LIN {X 0,Y 300.797,Z 338.167,A -85,B 0,C 180,E1 -24169.506,E2 -24169.506} C_VEL
LIN {X 0,Y 302.211,Z 343.381,A -85,B 0,C 180,E1 -24171.379,E2 -24171.379} C_VEL
LIN {X 0,Y 304.844,Z 348.124,A -85,B 0,C 180,E1 -24171.993,E2 -24171.993} C_VEL
LIN {X 0,Y 312.69,Z 363.044,A -85,B 0,C 180,E1 -24173.748,E2 -24173.748} C_VEL
LIN {X 0,Y 320.446,Z 379.712,A -85,B 0,C 180,E1 -24175.407,E2 -24175.407} C_VEL
LIN {X 0,Y 322.194,Z 383.758,A -85,B 0,C 180,E1 -24175.772,E2 -24175.772} C_VEL
LIN {X 0,Y 326.071,Z 409.314,A -85,B 0,C 180,E1 -24177.018,E2 -24177.018} C_VEL
LIN {X 0,Y 327.432,Z 420.163,A -85,B 0,C 180,E1 -24177.494,E2 -24177.494} C_VEL
LIN {X 0,Y 324.584,Z 482.925,A -85,B 0,C 180,E1 -24178.857,E2 -24178.857} C_VEL
LIN {X 0,Y 323.216,Z 497.454,A -85,B 0,C 180,E1 -24179.389,E2 -24179.389} C_VEL
LIN {X 0,Y 321.164,Z 510.847,A -85,B 0,C 180,E1 -24180.077,E2 -24180.077} C_VEL
LIN {X 0,Y 318.382,Z 524.837,A -85,B 0,C 180,E1 -24181.057,E2 -24181.057} C_VEL
LIN {X 0,Y 315.503,Z 537.338,A -85,B 0,C 180,E1 -24182.215,E2 -24182.215} C_VEL
LIN {X 0,Y 312.38,Z 548.887,A -85,B 0,C 180,E1 -24183.557,E2 -24183.557} C_VEL
LIN {X 0,Y 308.98,Z 560.643,A -85,B 0,C 180,E1 -24185.278,E2 -24185.278} C_VEL
LIN {X 0,Y 305.615,Z 570.588,A -85,B 0,C 180,E1 -24187.073,E2 -24187.073} C_VEL
LIN {X 0,Y 302.649,Z 579.143,A -85,B 0,C 180,E1 -24188.982,E2 -24188.982} C_VEL
LIN {X 0,Y 299.681,Z 587.381,A -85,B 0,C 180,E1 -24191.257,E2 -24191.257} C_VEL
LIN {X 0,Y 297.335,Z 594.052,A -85,B 0,C 180,E1 -24193.583,E2 -24193.583} C_VEL
LIN {X 0,Y 295.224,Z 600.025,A -85,B 0,C 180,E1 -24196.279,E2 -24196.279} C_VEL
LIN {X 0,Y 293.79,Z 604.467,A -85,B 0,C 180,E1 -24199.008,E2 -24199.008} C_VEL
LIN {X 0,Y 292.938,Z 607.496,A -85,B 0,C 180,E1 -24201.755,E2 -24201.755} C_VEL
LIN {X 0,Y 292.769,Z 609.197,A -85,B 0,C 180,E1 -24204.512,E2 -24204.512} C_VEL
LIN {X 0,Y 293.043,Z 609.861,A -85,B 0,C 180,E1 -24206.749,E2 -24206.749} C_VEL
LIN {X 0,Y 292.991,Z 613.677,A -85,B 0,C 180,E1 -24208.633,E2 -24208.633} C_VEL
LIN {X 0,Y 292.914,Z 615.958,A -85,B 0,C 180,E1 -24210.003,E2 -24210.003} C_VEL
LIN {X 0,Y 292.856,Z 617.841,A -85,B 0,C 180,E1 -24211.374,E2 -24211.374} C_VEL
LIN {X 0,Y 292.699,Z 620.456,A -85,B 0,C 180,E1 -24214.12,E2 -24214.12} C_VEL
LIN {X 0,Y 292.878,Z 621.675,A -85,B 0,C 180,E1 -24216.871,E2 -24216.871} C_VEL
LIN {X 0,Y 293.696,Z 621.539,A -85,B 0,C 180,E1 -24219.613,E2 -24219.613} C_VEL
LIN {X 0,Y 295.23,Z 620.064,A -85,B 0,C 180,E1 -24222.332,E2 -24222.332} C_VEL
LIN {X 0,Y 297.448,Z 617.232,A -85,B 0,C 180,E1 -24225.016,E2 -24225.016} C_VEL
LIN {X 0,Y 300.32,Z 613.003,A -85,B 0,C 180,E1 -24227.653,E2 -24227.653} C_VEL
LIN {X 0,Y 304.069,Z 607.239,A -85,B 0,C 180,E1 -24230.218,E2 -24230.218} C_VEL
LIN {X 0,Y 308.257,Z 599.867,A -85,B 0,C 180,E1 -24232.727,E2 -24232.727} C_VEL
LIN {X 0,Y 312.605,Z 591.846,A -85,B 0,C 180,E1 -24234.846,E2 -24234.846} C_VEL
LIN {X 0,Y 317.576,Z 581.993,A -85,B 0,C 180,E1 -24236.885,E2 -24236.885} C_VEL
LIN {X 0,Y 322.111,Z 571.917,A -85,B 0,C 180,E1 -24238.584,E2 -24238.584} C_VEL
LIN {X 0,Y 327.168,Z 559.76,A -85,B 0,C 180,E1 -24240.209,E2 -24240.209} C_VEL
LIN {X 0,Y 331.642,Z 547.568,A -85,B 0,C 180,E1 -24241.519,E2 -24241.519} C_VEL
LIN {X 0,Y 335.963,Z 534.106,A -85,B 0,C 180,E1 -24242.65,E2 -24242.65} C_VEL
LIN {X 0,Y 339.758,Z 520.179,A -85,B 0,C 180,E1 -24243.56,E2 -24243.56} C_VEL
LIN {X 0,Y 343.221,Z 504.513,A -85,B 0,C 180,E1 -24244.32,E2 -24244.32} C_VEL
LIN {X 0,Y 345.995,Z 486.463,A -85,B 0,C 180,E1 -24244.974,E2 -24244.974} C_VEL
LIN {X 0,Y 354.367,Z 425.402,A -85,B 0,C 180,E1 -24246.987,E2 -24246.987} C_VEL
LIN {X 0,Y 354.895,Z 409.778,A -85,B 0,C 180,E1 -24248.063,E2 -24248.063} C_VEL
LIN {X 0,Y 354.892,Z 404.222,A -85,B 0,C 180,E1 -24248.533,E2 -24248.533} C_VEL
LIN {X 0,Y 351.993,Z 398.922,A -85,B 0,C 180,E1 -24250.137,E2 -24250.137} C_VEL
LIN {X 0,Y 349.155,Z 394.154,A -85,B 0,C 180,E1 -24251.973,E2 -24251.973} C_VEL
LIN {X 0,Y 346.445,Z 389.926,A -85,B 0,C 180,E1 -24254.143,E2 -24254.143} C_VEL
LIN {X 0,Y 344.063,Z 386.653,A -85,B 0,C 180,E1 -24256.83,E2 -24256.83} C_VEL
LIN {X 0,Y 342.971,Z 385.018,A -85,B 0,C 180,E1 -24259.085,E2 -24259.085} C_VEL
LIN {X 0,Y 342.569,Z 384.877,A -85,B 0,C 180,E1 -24260.988,E2 -24260.988} C_VEL
LIN {X 0,Y 342.794,Z 385.856,A -85,B 0,C 180,E1 -24263.24,E2 -24263.24} C_VEL
LIN {X 0,Y 343.914,Z 388.274,A -85,B 0,C 180,E1 -24265.709,E2 -24265.709} C_VEL
LIN {X 0,Y 345.45,Z 391.168,A -85,B 0,C 180,E1 -24267.652,E2 -24267.652} C_VEL
LIN {X 0,Y 347.616,Z 395.463,A -85,B 0,C 180,E1 -24269.669,E2 -24269.669} C_VEL
LIN {X 0,Y 350.041,Z 400.682,A -85,B 0,C 180,E1 -24271.488,E2 -24271.488} C_VEL
LIN {X 0,Y 352.53,Z 406.284,A -85,B 0,C 180,E1 -24273.065,E2 -24273.065} C_VEL
LIN {X 0,Y 355.247,Z 413.527,A -85,B 0,C 180,E1 -24274.647,E2 -24274.647} C_VEL
LIN {X 0,Y 355.798,Z 415.257,A -85,B 0,C 180,E1 -24274.963,E2 -24274.963} C_VEL
LIN {X 0,Y 345.082,Z 491.977,A -85,B 0,C 180,E1 -24277.473,E2 -24277.473} C_VEL
LIN {X 0,Y 342.297,Z 506.53,A -85,B 0,C 180,E1 -24278.15,E2 -24278.15} C_VEL
LIN {X 0,Y 339.262,Z 519.363,A -85,B 0,C 180,E1 -24278.939,E2 -24278.939} C_VEL
LIN {X 0,Y 335.283,Z 533.245,A -85,B 0,C 180,E1 -24280.025,E2 -24280.025} C_VEL
LIN {X 0,Y 330.843,Z 546.376,A -85,B 0,C 180,E1 -24281.324,E2 -24281.324} C_VEL
LIN {X 0,Y 326.196,Z 558.349,A -85,B 0,C 180,E1 -24282.827,E2 -24282.827} C_VEL
LIN {X 0,Y 321.417,Z 569.249,A -85,B 0,C 180,E1 -24284.517,E2 -24284.517} C_VEL
LIN {X 0,Y 317.149,Z 578.141,A -85,B 0,C 180,E1 -24286.233,E2 -24286.233} C_VEL
LIN {X 0,Y 312.46,Z 587.071,A -85,B 0,C 180,E1 -24288.36,E2 -24288.36} C_VEL
LIN {X 0,Y 308.831,Z 593.256,A -85,B 0,C 180,E1 -24290.206,E2 -24290.206} C_VEL
LIN {X 0,Y 305.489,Z 598.43,A -85,B 0,C 180,E1 -24292.093,E2 -24292.093} C_VEL
LIN {X 0,Y 301.664,Z 603.858,A -85,B 0,C 180,E1 -24294.671,E2 -24294.671} C_VEL
LIN {X 0,Y 298.589,Z 607.736,A -85,B 0,C 180,E1 -24297.311,E2 -24297.311} C_VEL
LIN {X 0,Y 296.174,Z 610.172,A -85,B 0,C 180,E1 -24300,E2 -24300} C_VEL
LIN {X 0,Y 294.541,Z 611.221,A -85,B 0,C 180,E1 -24302.761,E2 -24302.761} C_VEL
LIN {X 0,Y 293.318,Z 610.914,A -85,B 0,C 180,E1 -24305.481,E2 -24305.481} C_VEL
LIN {X 0,Y 292.619,Z 609.217,A -85,B 0,C 180,E1 -24308.257,E2 -24308.257} C_VEL
LIN {X 0,Y 292.451,Z 606.082,A -85,B 0,C 180,E1 -24311.047,E2 -24311.047} C_VEL
LIN {X 0,Y 292.426,Z 601.359,A -85,B 0,C 180,E1 -24313.859,E2 -24313.859} C_VEL
LIN {X 0,Y 292.682,Z 596.611,A -85,B 0,C 180,E1 -24315.975,E2 -24315.975} C_VEL
LIN {X 0,Y 292.964,Z 589.602,A -85,B 0,C 180,E1 -24318.469,E2 -24318.469} C_VEL
LIN {X 0,Y 293.408,Z 582.124,A -85,B 0,C 180,E1 -24320.617,E2 -24320.617} C_VEL
LIN {X 0,Y 294.017,Z 572.971,A -85,B 0,C 180,E1 -24322.776,E2 -24322.776} C_VEL
LIN {X 0,Y 294.913,Z 561.779,A -85,B 0,C 180,E1 -24324.934,E2 -24324.934} C_VEL
LIN {X 0,Y 295.828,Z 550.441,A -85,B 0,C 180,E1 -24326.735,E2 -24326.735} C_VEL
LIN {X 0,Y 296.868,Z 538.133,A -85,B 0,C 180,E1 -24328.349,E2 -24328.349} C_VEL
LIN {X 0,Y 297.935,Z 524.592,A -85,B 0,C 180,E1 -24329.778,E2 -24329.778} C_VEL
LIN {X 0,Y 298.972,Z 509.581,A -85,B 0,C 180,E1 -24331.026,E2 -24331.026} C_VEL
LIN {X 0,Y 299.875,Z 494.673,A -85,B 0,C 180,E1 -24331.952,E2 -24331.952} C_VEL
LIN {X 0,Y 300.629,Z 479.252,A -85,B 0,C 180,E1 -24332.619,E2 -24332.619} C_VEL
LIN {X 0,Y 304.208,Z 387.346,A -85,B 0,C 180,E1 -24335.809,E2 -24335.809} C_VEL
LIN {X 0,Y 301.045,Z 356.735,A -85,B 0,C 180,E1 -24337.024,E2 -24337.024} C_VEL
LIN {X 0,Y 300.349,Z 346.328,A -85,B 0,C 180,E1 -24337.446,E2 -24337.446} C_VEL
LIN {X 0,Y 300.175,Z 343.352,A -85,B 0,C 180,E1 -24338.04,E2 -24338.04} C_VEL
LIN {X 0,Y 297.01,Z 327.627,A -85,B 0,C 180,E1 -24341.325,E2 -24341.325} C_VEL
LIN {X 0,Y 295.544,Z 320.23,A -85,B 0,C 180,E1 -24342.922,E2 -24342.922} C_VEL
LIN {X 0,Y 295.452,Z 320.238,A -85,B 0,C 180,E1 -24347.302,E2 -24347.302} C_VEL
LIN {X 0,Y 295.445,Z 320.237,A -85,B 0,C 180,E1 -24350.196,E2 -24350.196} C_VEL
LIN {X 0,Y 295.51,Z 320.231,A -85,B 0,C 180,E1 -24353.697,E2 -24353.697} C_VEL
LIN {X 0,Y 295.49,Z 320.226,A -85,B 0,C 180,E1 -24356.958,E2 -24356.958} C_VEL
LIN {X 0,Y 295.495,Z 320.228,A -85,B 0,C 180,E1 -24361.289,E2 -24361.289} C_VEL
LIN {X 0,Y 295.544,Z 320.228,A -85,B 0,C 180,E1 -24364.745,E2 -24364.745} C_VEL
LIN {X 0,Y 295.589,Z 320.223,A -85,B 0,C 180,E1 -24367.716,E2 -24367.716} C_VEL
LIN {X 0,Y 295.64,Z 320.215,A -85,B 0,C 180,E1 -24372.058,E2 -24372.058} C_VEL
LIN {X 0,Y 295.631,Z 320.212,A -85,B 0,C 180,E1 -24372.909,E2 -24372.909} C_VEL
LIN {X 0,Y 296.667,Z 323.105,A -85,B 0,C 180,E1 -24373.079,E2 -24373.079} C_VEL
LIN {X 0,Y 305.844,Z 343.561,A -85,B 0,C 180,E1 -24374.382,E2 -24374.382} C_VEL
LIN {X 0,Y 310.372,Z 356.722,A -85,B 0,C 180,E1 -24375.069,E2 -24375.069} C_VEL
LIN {X 0,Y 307.539,Z 451.607,A -85,B 0,C 180,E1 -24377.25,E2 -24377.25} C_VEL
LIN {X 0,Y 306.788,Z 465.849,A -85,B 0,C 180,E1 -24377.847,E2 -24377.847} C_VEL
LIN {X 0,Y 305.716,Z 479.602,A -85,B 0,C 180,E1 -24378.683,E2 -24378.683} C_VEL
LIN {X 0,Y 304.431,Z 492.441,A -85,B 0,C 180,E1 -24379.725,E2 -24379.725} C_VEL
LIN {X 0,Y 302.99,Z 503.539,A -85,B 0,C 180,E1 -24380.852,E2 -24380.852} C_VEL
LIN {X 0,Y 301.227,Z 515.227,A -85,B 0,C 180,E1 -24382.313,E2 -24382.313} C_VEL
LIN {X 0,Y 299.781,Z 525.862,A -85,B 0,C 180,E1 -24383.961,E2 -24383.961} C_VEL
LIN {X 0,Y 298.014,Z 536.451,A -85,B 0,C 180,E1 -24385.953,E2 -24385.953} C_VEL
LIN {X 0,Y 296.649,Z 545.177,A -85,B 0,C 180,E1 -24387.967,E2 -24387.967} C_VEL
LIN {X 0,Y 295.166,Z 553.586,A -85,B 0,C 180,E1 -24390.337,E2 -24390.337} C_VEL
LIN {X 0,Y 294.481,Z 560.307,A -85,B 0,C 180,E1 -24392.723,E2 -24392.723} C_VEL
LIN {X 0,Y 293.842,Z 564.964,A -85,B 0,C 180,E1 -24394.782,E2 -24394.782} C_VEL
LIN {X 0,Y 293.151,Z 569.825,A -85,B 0,C 180,E1 -24397.548,E2 -24397.548} C_VEL
LIN {X 0,Y 292.981,Z 572.446,A -85,B 0,C 180,E1 -24399.63,E2 -24399.63} C_VEL
LIN {X 0,Y 292.991,Z 574.75,A -85,B 0,C 180,E1 -24402.421,E2 -24402.421} C_VEL
LIN {X 0,Y 293.267,Z 575.703,A -85,B 0,C 180,E1 -24405.228,E2 -24405.228} C_VEL
LIN {X 0,Y 293.998,Z 575.297,A -85,B 0,C 180,E1 -24408.039,E2 -24408.039} C_VEL
LIN {X 0,Y 295.098,Z 573.519,A -85,B 0,C 180,E1 -24410.853,E2 -24410.853} C_VEL
LIN {X 0,Y 296.806,Z 570.267,A -85,B 0,C 180,E1 -24413.649,E2 -24413.649} C_VEL
LIN {X 0,Y 298.986,Z 565.44,A -85,B 0,C 180,E1 -24416.427,E2 -24416.427} C_VEL
LIN {X 0,Y 301.008,Z 560.725,A -85,B 0,C 180,E1 -24418.488,E2 -24418.488} C_VEL
LIN {X 0,Y 303.824,Z 553.8,A -85,B 0,C 180,E1 -24420.857,E2 -24420.857} C_VEL
LIN {X 0,Y 306.53,Z 546.503,A -85,B 0,C 180,E1 -24422.864,E2 -24422.864} C_VEL
LIN {X 0,Y 309.598,Z 537.649,A -85,B 0,C 180,E1 -24424.834,E2 -24424.834} C_VEL
LIN {X 0,Y 312.693,Z 527.837,A -85,B 0,C 180,E1 -24426.608,E2 -24426.608} C_VEL
LIN {X 0,Y 315.695,Z 517.031,A -85,B 0,C 180,E1 -24428.2,E2 -24428.2} C_VEL
LIN {X 0,Y 318.559,Z 505.159,A -85,B 0,C 180,E1 -24429.612,E2 -24429.612} C_VEL
LIN {X 0,Y 321.196,Z 491.982,A -85,B 0,C 180,E1 -24430.856,E2 -24430.856} C_VEL
LIN {X 0,Y 323.29,Z 478.09,A -85,B 0,C 180,E1 -24431.876,E2 -24431.876} C_VEL
LIN {X 0,Y 324.931,Z 464.176,A -85,B 0,C 180,E1 -24432.608,E2 -24432.608} C_VEL
LIN {X 0,Y 325.962,Z 451.27,A -85,B 0,C 180,E1 -24433.075,E2 -24433.075} C_VEL
LIN {X 0,Y 329.077,Z 378.605,A -85,B 0,C 180,E1 -24434.666,E2 -24434.666} C_VEL
LIN {X 0,Y 321.686,Z 362.958,A -85,B 0,C 180,E1 -24436.139,E2 -24436.139} C_VEL
LIN {X 0,Y 315.094,Z 350.798,A -85,B 0,C 180,E1 -24437.49,E2 -24437.49} C_VEL
LIN {X 0,Y 306.413,Z 337.106,A -85,B 0,C 180,E1 -24439.334,E2 -24439.334} C_VEL
LIN {X 0,Y 300.748,Z 328.88,A -85,B 0,C 180,E1 -24440.607,E2 -24440.607} C_VEL
LIN {X 0,Y 298.582,Z 325.449,A -85,B 0,C 180,E1 -24441.125,E2 -24441.125} C_VEL
LIN {X 0,Y 296.267,Z 322.728,A -85,B 0,C 180,E1 -24441.659,E2 -24441.659} C_VEL
LIN {X 0,Y 295.501,Z 320.229,A -85,B 0,C 180,E1 -24441.908,E2 -24441.908} C_VEL
LIN {X 0,Y 295.464,Z 320.215,A -85,B 0,C 180,E1 -24446.064,E2 -24446.064} C_VEL
LIN {X 0,Y 295.486,Z 320.231,A -85,B 0,C 180,E1 -24450.145,E2 -24450.145} C_VEL
LIN {X 0,Y 295.534,Z 320.229,A -85,B 0,C 180,E1 -24454.232,E2 -24454.232} C_VEL
LIN {X 0,Y 295.565,Z 320.215,A -85,B 0,C 180,E1 -24457.717,E2 -24457.717} C_VEL
LIN {X 0,Y 295.598,Z 320.21,A -85,B 0,C 180,E1 -24462.059,E2 -24462.059} C_VEL
LIN {X 0,Y 295.704,Z 320.19,A -85,B 0,C 180,E1 -24466.298,E2 -24466.298} C_VEL
LIN {X 0,Y 295.767,Z 320.183,A -85,B 0,C 180,E1 -24470.458,E2 -24470.458} C_VEL
LIN {X 0,Y 295.98,Z 320.175,A -85,B 0,C 180,E1 -24473.652,E2 -24473.652} C_VEL
LIN {X 0,Y 295.931,Z 320.172,A -85,B 0,C 180,E1 -24474.741,E2 -24474.741} C_VEL
LIN {X 0,Y 295.298,Z 320.24,A -85,B 0,C 180,E1 -24475.878,E2 -24475.878} C_VEL
LIN {X 0,Y 292.497,Z 320.595,A -85,B 0,C 180,E1 -24477.732,E2 -24477.732} C_VEL
LIN {X 0,Y 290.109,Z 320.907,A -85,B 0,C 180,E1 -24479.236,E2 -24479.236} C_VEL
LIN {X 0,Y 289.085,Z 321.022,A -85,B 0,C 180,E1 -24480.401,E2 -24480.401} C_VEL
LIN {X 0,Y 289.003,Z 321.026,A -85,B 0,C 180,E1 -24480.795,E2 -24480.795} C_VEL
LIN {X 0,Y 288.971,Z 321.045,A -85,B 0,C 180,E1 -24484.17,E2 -24484.17} C_VEL
LIN {X 0,Y 288.857,Z 321.038,A -85,B 0,C 180,E1 -24486.964,E2 -24486.964} C_VEL
LIN {X 0,Y 288.675,Z 321.071,A -85,B 0,C 180,E1 -24491.193,E2 -24491.193} C_VEL
LIN {X 0,Y 288.684,Z 321.07,A -85,B 0,C 180,E1 -24494.042,E2 -24494.042} C_VEL
LIN {X 0,Y 288.57,Z 321.083,A -85,B 0,C 180,E1 -24498.814,E2 -24498.814} C_VEL
LIN {X 0,Y 288.493,Z 321.091,A -85,B 0,C 180,E1 -24502.859,E2 -24502.859} C_VEL
LIN {X 0,Y 288.479,Z 321.095,A -85,B 0,C 180,E1 -24506.063,E2 -24506.063} C_VEL
LIN {X 0,Y 288.447,Z 321.1,A -85,B 0,C 180,E1 -24510.661,E2 -24510.661} C_VEL
LIN {X 0,Y 288.455,Z 321.075,A -85,B 0,C 180,E1 -24514.357,E2 -24514.357} C_VEL
LIN {X 0,Y 288.484,Z 321.076,A -85,B 0,C 180,E1 -24517.373,E2 -24517.373} C_VEL
LIN {X 0,Y 288.52,Z 321.266,A -85,B 0,C 180,E1 -24520.841,E2 -24520.841} C_VEL
LIN {X 0,Y 291.2,Z 330.037,A -85,B 0,C 180,E1 -24524.886,E2 -24524.886} C_VEL
LIN {X 0,Y 293.848,Z 339.179,A -85,B 0,C 180,E1 -24528.664,E2 -24528.664} C_VEL
LIN {X 0,Y 294.769,Z 342.618,A -85,B 0,C 180,E1 -24529.975,E2 -24529.975} C_VEL
LIN {X 0,Y 297.416,Z 347.373,A -85,B 0,C 180,E1 -24530.635,E2 -24530.635} C_VEL
LIN {X 0,Y 302.135,Z 355.948,A -85,B 0,C 180,E1 -24531.77,E2 -24531.77} C_VEL
LIN {X 0,Y 307.935,Z 366.963,A -85,B 0,C 180,E1 -24533.1,E2 -24533.1} C_VEL
LIN {X 0,Y 316.042,Z 384.747,A -85,B 0,C 180,E1 -24534.904,E2 -24534.904} C_VEL
LIN {X 0,Y 316.961,Z 387.009,A -85,B 0,C 180,E1 -24535.106,E2 -24535.106} C_VEL
LIN {X 0,Y 320.494,Z 411.032,A -85,B 0,C 180,E1 -24536.3,E2 -24536.3} C_VEL
LIN {X 0,Y 321.741,Z 421.145,A -85,B 0,C 180,E1 -24536.757,E2 -24536.757} C_VEL
LIN {X 0,Y 318.823,Z 482.959,A -85,B 0,C 180,E1 -24538.121,E2 -24538.121} C_VEL
LIN {X 0,Y 317.373,Z 497.579,A -85,B 0,C 180,E1 -24538.67,E2 -24538.67} C_VEL
LIN {X 0,Y 315.072,Z 511.951,A -85,B 0,C 180,E1 -24539.438,E2 -24539.438} C_VEL
LIN {X 0,Y 312.597,Z 523.859,A -85,B 0,C 180,E1 -24540.284,E2 -24540.284} C_VEL
LIN {X 0,Y 309.625,Z 536.466,A -85,B 0,C 180,E1 -24541.456,E2 -24541.456} C_VEL
LIN {X 0,Y 306.392,Z 547.981,A -85,B 0,C 180,E1 -24542.796,E2 -24542.796} C_VEL
LIN {X 0,Y 303.086,Z 559.192,A -85,B 0,C 180,E1 -24544.445,E2 -24544.445} C_VEL
LIN {X 0,Y 299.679,Z 569.096,A -85,B 0,C 180,E1 -24546.226,E2 -24546.226} C_VEL
LIN {X 0,Y 296.488,Z 577.824,A -85,B 0,C 180,E1 -24548.159,E2 -24548.159} C_VEL
LIN {X 0,Y 293.313,Z 586.236,A -85,B 0,C 180,E1 -24550.472,E2 -24550.472} C_VEL
LIN {X 0,Y 291.123,Z 592.138,A -85,B 0,C 180,E1 -24552.501,E2 -24552.501} C_VEL
LIN {X 0,Y 288.819,Z 598.498,A -85,B 0,C 180,E1 -24555.251,E2 -24555.251} C_VEL
LIN {X 0,Y 287.133,Z 603.27,A -85,B 0,C 180,E1 -24558.036,E2 -24558.036} C_VEL
LIN {X 0,Y 286.251,Z 605.853,A -85,B 0,C 180,E1 -24560.141,E2 -24560.141} C_VEL
LIN {X 0,Y 285.656,Z 608.156,A -85,B 0,C 180,E1 -24562.961,E2 -24562.961} C_VEL
LIN {X 0,Y 285.814,Z 609.158,A -85,B 0,C 180,E1 -24565.787,E2 -24565.787} C_VEL
LIN {X 0,Y 285.986,Z 609.357,A -85,B 0,C 180,E1 -24566.932,E2 -24566.932} C_VEL
LIN {X 0,Y 285.926,Z 614.016,A -85,B 0,C 180,E1 -24569.302,E2 -24569.302} C_VEL
LIN {X 0,Y 285.81,Z 617.126,A -85,B 0,C 180,E1 -24571.408,E2 -24571.408} C_VEL
LIN {X 0,Y 285.62,Z 619.941,A -85,B 0,C 180,E1 -24574.222,E2 -24574.222} C_VEL
LIN {X 0,Y 285.81,Z 621.356,A -85,B 0,C 180,E1 -24577.042,E2 -24577.042} C_VEL
LIN {X 0,Y 286.694,Z 621.438,A -85,B 0,C 180,E1 -24579.851,E2 -24579.851} C_VEL
LIN {X 0,Y 288.302,Z 620.193,A -85,B 0,C 180,E1 -24582.634,E2 -24582.634} C_VEL
LIN {X 0,Y 290.678,Z 617.546,A -85,B 0,C 180,E1 -24585.446,E2 -24585.446} C_VEL
LIN {X 0,Y 293.616,Z 613.677,A -85,B 0,C 180,E1 -24588.07,E2 -24588.07} C_VEL
LIN {X 0,Y 296.423,Z 609.715,A -85,B 0,C 180,E1 -24590.041,E2 -24590.041} C_VEL
LIN {X 0,Y 300.744,Z 603.088,A -85,B 0,C 180,E1 -24592.603,E2 -24592.603} C_VEL
LIN {X 0,Y 305.017,Z 595.837,A -85,B 0,C 180,E1 -24594.781,E2 -24594.781} C_VEL
LIN {X 0,Y 309.944,Z 587,A -85,B 0,C 180,E1 -24596.874,E2 -24596.874} C_VEL
LIN {X 0,Y 315.313,Z 576.224,A -85,B 0,C 180,E1 -24598.895,E2 -24598.895} C_VEL
LIN {X 0,Y 320.451,Z 565.032,A -85,B 0,C 180,E1 -24600.547,E2 -24600.547} C_VEL
LIN {X 0,Y 325.459,Z 552.766,A -85,B 0,C 180,E1 -24602.007,E2 -24602.007} C_VEL
LIN {X 0,Y 329.801,Z 540.581,A -85,B 0,C 180,E1 -24603.157,E2 -24603.157} C_VEL
LIN {X 0,Y 334.437,Z 525.531,A -85,B 0,C 180,E1 -24604.257,E2 -24604.257} C_VEL
LIN {X 0,Y 337.971,Z 511.719,A -85,B 0,C 180,E1 -24605.02,E2 -24605.02} C_VEL
LIN {X 0,Y 341.055,Z 495.588,A -85,B 0,C 180,E1 -24605.693,E2 -24605.693} C_VEL
LIN {X 0,Y 350.969,Z 427.139,A -85,B 0,C 180,E1 -24607.962,E2 -24607.962} C_VEL
LIN {X 0,Y 351.68,Z 411.85,A -85,B 0,C 180,E1 -24609.034,E2 -24609.034} C_VEL
LIN {X 0,Y 351.667,Z 409.048,A -85,B 0,C 180,E1 -24609.298,E2 -24609.298} C_VEL
LIN {X 0,Y 348.159,Z 402.533,A -85,B 0,C 180,E1 -24611.481,E2 -24611.481} C_VEL
LIN {X 0,Y 345.228,Z 397.709,A -85,B 0,C 180,E1 -24613.748,E2 -24613.748} C_VEL
LIN {X 0,Y 343.498,Z 395.172,A -85,B 0,C 180,E1 -24615.483,E2 -24615.483} C_VEL
LIN {X 0,Y 341.777,Z 392.491,A -85,B 0,C 180,E1 -24618.134,E2 -24618.134} C_VEL
LIN {X 0,Y 341.305,Z 391.878,A -85,B 0,C 180,E1 -24619.409,E2 -24619.409} C_VEL
LIN {X 0,Y 340.993,Z 391.879,A -85,B 0,C 180,E1 -24621.316,E2 -24621.316} C_VEL
LIN {X 0,Y 341.332,Z 393.124,A -85,B 0,C 180,E1 -24623.65,E2 -24623.65} C_VEL
LIN {X 0,Y 342.426,Z 395.587,A -85,B 0,C 180,E1 -24625.902,E2 -24625.902} C_VEL
LIN {X 0,Y 343.605,Z 397.91,A -85,B 0,C 180,E1 -24627.436,E2 -24627.436} C_VEL
LIN {X 0,Y 345.579,Z 402.063,A -85,B 0,C 180,E1 -24629.381,E2 -24629.381} C_VEL
LIN {X 0,Y 347.724,Z 407.035,A -85,B 0,C 180,E1 -24631.117,E2 -24631.117} C_VEL
LIN {X 0,Y 349.782,Z 411.933,A -85,B 0,C 180,E1 -24632.523,E2 -24632.523} C_VEL
LIN {X 0,Y 352.218,Z 418.848,A -85,B 0,C 180,E1 -24634.055,E2 -24634.055} C_VEL
LIN {X 0,Y 341.436,Z 492.23,A -85,B 0,C 180,E1 -24636.46,E2 -24636.46} C_VEL
LIN {X 0,Y 338.396,Z 507.306,A -85,B 0,C 180,E1 -24637.163,E2 -24637.163} C_VEL
LIN {X 0,Y 335.364,Z 519.52,A -85,B 0,C 180,E1 -24637.917,E2 -24637.917} C_VEL
LIN {X 0,Y 331.412,Z 532.712,A -85,B 0,C 180,E1 -24638.943,E2 -24638.943} C_VEL
LIN {X 0,Y 326.679,Z 546.19,A -85,B 0,C 180,E1 -24640.263,E2 -24640.263} C_VEL
LIN {X 0,Y 322.237,Z 557.207,A -85,B 0,C 180,E1 -24641.628,E2 -24641.628} C_VEL
LIN {X 0,Y 317.17,Z 568.297,A -85,B 0,C 180,E1 -24643.316,E2 -24643.316} C_VEL
LIN {X 0,Y 311.931,Z 578.669,A -85,B 0,C 180,E1 -24645.313,E2 -24645.313} C_VEL
LIN {X 0,Y 306.938,Z 587.578,A -85,B 0,C 180,E1 -24647.479,E2 -24647.479} C_VEL
LIN {X 0,Y 303.122,Z 593.711,A -85,B 0,C 180,E1 -24649.347,E2 -24649.347} C_VEL
LIN {X 0,Y 299.597,Z 598.81,A -85,B 0,C 180,E1 -24651.259,E2 -24651.259} C_VEL
LIN {X 0,Y 296.157,Z 603.344,A -85,B 0,C 180,E1 -24653.408,E2 -24653.408} C_VEL
LIN {X 0,Y 292.946,Z 607.163,A -85,B 0,C 180,E1 -24655.887,E2 -24655.887} C_VEL
LIN {X 0,Y 290.12,Z 609.911,A -85,B 0,C 180,E1 -24658.617,E2 -24658.617} C_VEL
LIN {X 0,Y 288.146,Z 611.271,A -85,B 0,C 180,E1 -24661.393,E2 -24661.393} C_VEL
LIN {X 0,Y 286.718,Z 611.295,A -85,B 0,C 180,E1 -24664.203,E2 -24664.203} C_VEL
LIN {X 0,Y 285.743,Z 609.949,A -85,B 0,C 180,E1 -24667.04,E2 -24667.04} C_VEL
LIN {X 0,Y 285.4,Z 607.188,A -85,B 0,C 180,E1 -24669.892,E2 -24669.892} C_VEL
LIN {X 0,Y 285.3,Z 604.08,A -85,B 0,C 180,E1 -24672.045,E2 -24672.045} C_VEL
LIN {X 0,Y 285.384,Z 600.038,A -85,B 0,C 180,E1 -24674.208,E2 -24674.208} C_VEL
LIN {X 0,Y 285.636,Z 595.097,A -85,B 0,C 180,E1 -24676.332,E2 -24676.332} C_VEL
LIN {X 0,Y 285.991,Z 587.465,A -85,B 0,C 180,E1 -24678.936,E2 -24678.936} C_VEL
LIN {X 0,Y 286.496,Z 579.493,A -85,B 0,C 180,E1 -24681.138,E2 -24681.138} C_VEL
LIN {X 0,Y 287.123,Z 569.762,A -85,B 0,C 180,E1 -24683.355,E2 -24683.355} C_VEL
LIN {X 0,Y 288.023,Z 558.97,A -85,B 0,C 180,E1 -24685.38,E2 -24685.38} C_VEL
LIN {X 0,Y 289.01,Z 547.131,A -85,B 0,C 180,E1 -24687.203,E2 -24687.203} C_VEL
LIN {X 0,Y 290.123,Z 533.856,A -85,B 0,C 180,E1 -24688.872,E2 -24688.872} C_VEL
LIN {X 0,Y 291.149,Z 520.473,A -85,B 0,C 180,E1 -24690.227,E2 -24690.227} C_VEL
LIN {X 0,Y 292.111,Z 506.469,A -85,B 0,C 180,E1 -24691.335,E2 -24691.335} C_VEL
LIN {X 0,Y 293.096,Z 490.523,A -85,B 0,C 180,E1 -24692.274,E2 -24692.274} C_VEL
LIN {X 0,Y 293.959,Z 468.714,A -85,B 0,C 180,E1 -24693.131,E2 -24693.131} C_VEL
LIN {X 0,Y 297.198,Z 387.774,A -85,B 0,C 180,E1 -24696.028,E2 -24696.028} C_VEL
LIN {X 0,Y 293.975,Z 356.014,A -85,B 0,C 180,E1 -24697.32,E2 -24697.32} C_VEL
LIN {X 0,Y 293.437,Z 346.313,A -85,B 0,C 180,E1 -24697.744,E2 -24697.744} C_VEL
LIN {X 0,Y 290.656,Z 331.948,A -85,B 0,C 180,E1 -24700.779,E2 -24700.779} C_VEL
LIN {X 0,Y 288.517,Z 321.104,A -85,B 0,C 180,E1 -24703.135,E2 -24703.135} C_VEL
LIN {X 0,Y 288.403,Z 321.116,A -85,B 0,C 180,E1 -24707.15,E2 -24707.15} C_VEL
LIN {X 0,Y 288.4,Z 321.116,A -85,B 0,C 180,E1 -24711.004,E2 -24711.004} C_VEL
LIN {X 0,Y 288.422,Z 321.107,A -85,B 0,C 180,E1 -24714.345,E2 -24714.345} C_VEL
LIN {X 0,Y 288.433,Z 321.112,A -85,B 0,C 180,E1 -24718.207,E2 -24718.207} C_VEL
LIN {X 0,Y 288.476,Z 321.099,A -85,B 0,C 180,E1 -24722.523,E2 -24722.523} C_VEL
LIN {X 0,Y 288.466,Z 321.11,A -85,B 0,C 180,E1 -24725.617,E2 -24725.617} C_VEL
LIN {X 0,Y 288.514,Z 321.104,A -85,B 0,C 180,E1 -24728.641,E2 -24728.641} C_VEL
LIN {X 0,Y 288.598,Z 321.09,A -85,B 0,C 180,E1 -24732.28,E2 -24732.28} C_VEL
LIN {X 0,Y 289.663,Z 324.032,A -85,B 0,C 180,E1 -24732.467,E2 -24732.467} C_VEL
LIN {X 0,Y 299.147,Z 344.931,A -85,B 0,C 180,E1 -24733.863,E2 -24733.863} C_VEL
LIN {X 0,Y 303.714,Z 357.761,A -85,B 0,C 180,E1 -24734.569,E2 -24734.569} C_VEL
LIN {X 0,Y 300.953,Z 451.074,A -85,B 0,C 180,E1 -24736.752,E2 -24736.752} C_VEL
LIN {X 0,Y 300.112,Z 465.674,A -85,B 0,C 180,E1 -24737.358,E2 -24737.358} C_VEL
LIN {X 0,Y 299.123,Z 478.993,A -85,B 0,C 180,E1 -24738.174,E2 -24738.174} C_VEL
LIN {X 0,Y 297.88,Z 491.182,A -85,B 0,C 180,E1 -24739.154,E2 -24739.154} C_VEL
LIN {X 0,Y 296.416,Z 502.592,A -85,B 0,C 180,E1 -24740.304,E2 -24740.304} C_VEL
LIN {X 0,Y 294.57,Z 514.523,A -85,B 0,C 180,E1 -24741.794,E2 -24741.794} C_VEL
LIN {X 0,Y 293.043,Z 525.348,A -85,B 0,C 180,E1 -24743.478,E2 -24743.478} C_VEL
LIN {X 0,Y 291.527,Z 534.46,A -85,B 0,C 180,E1 -24745.173,E2 -24745.173} C_VEL
LIN {X 0,Y 289.955,Z 543.602,A -85,B 0,C 180,E1 -24747.227,E2 -24747.227} C_VEL
LIN {X 0,Y 288.583,Z 551.237,A -85,B 0,C 180,E1 -24749.301,E2 -24749.301} C_VEL
LIN {X 0,Y 287.813,Z 557.557,A -85,B 0,C 180,E1 -24751.391,E2 -24751.391} C_VEL
LIN {X 0,Y 287.156,Z 562.775,A -85,B 0,C 180,E1 -24753.493,E2 -24753.493} C_VEL
LIN {X 0,Y 286.337,Z 568.329,A -85,B 0,C 180,E1 -24756.316,E2 -24756.316} C_VEL
LIN {X 0,Y 285.958,Z 571.43,A -85,B 0,C 180,E1 -24758.448,E2 -24758.448} C_VEL
LIN {X 0,Y 285.914,Z 574.494,A -85,B 0,C 180,E1 -24761.496,E2 -24761.496} C_VEL
LIN {X 0,Y 286.026,Z 575.882,A -85,B 0,C 180,E1 -24764.171,E2 -24764.171} C_VEL
LIN {X 0,Y 286.62,Z 576.071,A -85,B 0,C 180,E1 -24767.049,E2 -24767.049} C_VEL
LIN {X 0,Y 287.576,Z 574.891,A -85,B 0,C 180,E1 -24769.934,E2 -24769.934} C_VEL
LIN {X 0,Y 289.128,Z 572.273,A -85,B 0,C 180,E1 -24772.802,E2 -24772.802} C_VEL
LIN {X 0,Y 291.197,Z 568.15,A -85,B 0,C 180,E1 -24775.652,E2 -24775.652} C_VEL
LIN {X 0,Y 293.811,Z 562.39,A -85,B 0,C 180,E1 -24778.472,E2 -24778.472} C_VEL
LIN {X 0,Y 296.64,Z 555.823,A -85,B 0,C 180,E1 -24780.898,E2 -24780.898} C_VEL
LIN {X 0,Y 299.885,Z 547.587,A -85,B 0,C 180,E1 -24783.286,E2 -24783.286} C_VEL
LIN {X 0,Y 303.037,Z 538.876,A -85,B 0,C 180,E1 -24785.295,E2 -24785.295} C_VEL
LIN {X 0,Y 305.936,Z 530.186,A -85,B 0,C 180,E1 -24786.937,E2 -24786.937} C_VEL
LIN {X 0,Y 309.307,Z 518.619,A -85,B 0,C 180,E1 -24788.72,E2 -24788.72} C_VEL
LIN {X 0,Y 312.387,Z 506.521,A -85,B 0,C 180,E1 -24790.204,E2 -24790.204} C_VEL
LIN {X 0,Y 314.997,Z 494.177,A -85,B 0,C 180,E1 -24791.412,E2 -24791.412} C_VEL
LIN {X 0,Y 317.142,Z 480.787,A -85,B 0,C 180,E1 -24792.45,E2 -24792.45} C_VEL
LIN {X 0,Y 318.992,Z 466.368,A -85,B 0,C 180,E1 -24793.262,E2 -24793.262} C_VEL
LIN {X 0,Y 320.198,Z 452.251,A -85,B 0,C 180,E1 -24793.802,E2 -24793.802} C_VEL
LIN {X 0,Y 323.423,Z 380.829,A -85,B 0,C 180,E1 -24795.384,E2 -24795.384} C_VEL
LIN {X 0,Y 316.028,Z 365.317,A -85,B 0,C 180,E1 -24796.915,E2 -24796.915} C_VEL
LIN {X 0,Y 310.501,Z 355.137,A -85,B 0,C 180,E1 -24798.093,E2 -24798.093} C_VEL
LIN {X 0,Y 302.397,Z 342.254,A -85,B 0,C 180,E1 -24799.873,E2 -24799.873} C_VEL
LIN {X 0,Y 296.243,Z 333.323,A -85,B 0,C 180,E1 -24801.305,E2 -24801.305} C_VEL
LIN {X 0,Y 294.19,Z 330.234,A -85,B 0,C 180,E1 -24801.808,E2 -24801.808} C_VEL
LIN {X 0,Y 292.018,Z 327.194,A -85,B 0,C 180,E1 -24802.345,E2 -24802.345} C_VEL
LIN {X 0,Y 291.225,Z 325.908,A -85,B 0,C 180,E1 -24802.551,E2 -24802.551} C_VEL
LIN {X 0,Y 289.971,Z 324.694,A -85,B 0,C 180,E1 -24802.851,E2 -24802.851} C_VEL
LIN {X 0,Y 288.642,Z 322.163,A -85,B 0,C 180,E1 -24803.218,E2 -24803.218} C_VEL
LIN {X 0,Y 288.433,Z 321.081,A -85,B 0,C 180,E1 -24803.328,E2 -24803.328} C_VEL
LIN {X 0,Y 288.427,Z 321.091,A -85,B 0,C 180,E1 -24806.044,E2 -24806.044} C_VEL
LIN {X 0,Y 288.437,Z 321.103,A -85,B 0,C 180,E1 -24809.338,E2 -24809.338} C_VEL
LIN {X 0,Y 288.463,Z 321.097,A -85,B 0,C 180,E1 -24812.525,E2 -24812.525} C_VEL
LIN {X 0,Y 288.464,Z 321.102,A -85,B 0,C 180,E1 -24815.62,E2 -24815.62} C_VEL
LIN {X 0,Y 288.488,Z 321.108,A -85,B 0,C 180,E1 -24818.642,E2 -24818.642} C_VEL
LIN {X 0,Y 288.551,Z 321.084,A -85,B 0,C 180,E1 -24821.605,E2 -24821.605} C_VEL
LIN {X 0,Y 288.641,Z 321.069,A -85,B 0,C 180,E1 -24826.073,E2 -24826.073} C_VEL
LIN {X 0,Y 288.718,Z 321.062,A -85,B 0,C 180,E1 -24830.222,E2 -24830.222} C_VEL
LIN {X 0,Y 288.887,Z 321.055,A -85,B 0,C 180,E1 -24834.434,E2 -24834.434} C_VEL
LIN {X 0,Y 288.934,Z 321.033,A -85,B 0,C 180,E1 -24837.221,E2 -24837.221} C_VEL
LIN {X 0,Y 289.003,Z 321.026,A -85,B 0,C 180,E1 -24840.795,E2 -24840.795} C_VEL
LIN {X 0,Y 288.342,Z 321.106,A -85,B 0,C 180,E1 -24841.958,E2 -24841.958} C_VEL
LIN {X 0,Y 285.487,Z 321.476,A -85,B 0,C 180,E1 -24843.85,E2 -24843.85} C_VEL
LIN {X 0,Y 283.028,Z 321.782,A -85,B 0,C 180,E1 -24845.386,E2 -24845.386} C_VEL
LIN {X 0,Y 281.925,Z 321.905,A -85,B 0,C 180,E1 -24846.577,E2 -24846.577} C_VEL
LIN {X 0,Y 281.809,Z 321.916,A -85,B 0,C 180,E1 -24846.981,E2 -24846.981} C_VEL
LIN {X 0,Y 281.618,Z 321.945,A -85,B 0,C 180,E1 -24851.477,E2 -24851.477} C_VEL
LIN {X 0,Y 281.604,Z 321.957,A -85,B 0,C 180,E1 -24854.403,E2 -24854.403} C_VEL
LIN {X 0,Y 281.517,Z 321.964,A -85,B 0,C 180,E1 -24859.02,E2 -24859.02} C_VEL
LIN {X 0,Y 281.432,Z 321.976,A -85,B 0,C 180,E1 -24863.467,E2 -24863.467} C_VEL
LIN {X 0,Y 281.408,Z 321.975,A -85,B 0,C 180,E1 -24866.618,E2 -24866.618} C_VEL
LIN {X 0,Y 281.384,Z 321.982,A -85,B 0,C 180,E1 -24869.858,E2 -24869.858} C_VEL
LIN {X 0,Y 281.381,Z 321.979,A -85,B 0,C 180,E1 -24873.206,E2 -24873.206} C_VEL
LIN {X 0,Y 281.447,Z 321.949,A -85,B 0,C 180,E1 -24877.22,E2 -24877.22} C_VEL
LIN {X 0,Y 281.468,Z 322.099,A -85,B 0,C 180,E1 -24879.46,E2 -24879.46} C_VEL
LIN {X 0,Y 284.15,Z 330.711,A -85,B 0,C 180,E1 -24883.647,E2 -24883.647} C_VEL
LIN {X 0,Y 286.486,Z 338.767,A -85,B 0,C 180,E1 -24887.179,E2 -24887.179} C_VEL
LIN {X 0,Y 287.478,Z 342.144,A -85,B 0,C 180,E1 -24888.501,E2 -24888.501} C_VEL
LIN {X 0,Y 289.985,Z 346.644,A -85,B 0,C 180,E1 -24889.172,E2 -24889.172} C_VEL
LIN {X 0,Y 294.715,Z 354.806,A -85,B 0,C 180,E1 -24890.377,E2 -24890.377} C_VEL
LIN {X 0,Y 301.598,Z 367.687,A -85,B 0,C 180,E1 -24892.05,E2 -24892.05} C_VEL
LIN {X 0,Y 308.041,Z 381.411,A -85,B 0,C 180,E1 -24893.559,E2 -24893.559} C_VEL
LIN {X 0,Y 311.778,Z 390.361,A -85,B 0,C 180,E1 -24894.42,E2 -24894.42} C_VEL
LIN {X 0,Y 315.111,Z 413.914,A -85,B 0,C 180,E1 -24895.612,E2 -24895.612} C_VEL
LIN {X 0,Y 316.106,Z 422.6,A -85,B 0,C 180,E1 -24896.006,E2 -24896.006} C_VEL
LIN {X 0,Y 313.195,Z 482.218,A -85,B 0,C 180,E1 -24897.336,E2 -24897.336} C_VEL
LIN {X 0,Y 311.784,Z 496.199,A -85,B 0,C 180,E1 -24897.853,E2 -24897.853} C_VEL
LIN {X 0,Y 309.625,Z 509.697,A -85,B 0,C 180,E1 -24898.556,E2 -24898.556} C_VEL
LIN {X 0,Y 306.893,Z 522.877,A -85,B 0,C 180,E1 -24899.485,E2 -24899.485} C_VEL
LIN {X 0,Y 303.808,Z 535.594,A -85,B 0,C 180,E1 -24900.668,E2 -24900.668} C_VEL
LIN {X 0,Y 300.126,Z 548.355,A -85,B 0,C 180,E1 -24902.18,E2 -24902.18} C_VEL
LIN {X 0,Y 297.008,Z 558.497,A -85,B 0,C 180,E1 -24903.701,E2 -24903.701} C_VEL
LIN {X 0,Y 293.198,Z 569.229,A -85,B 0,C 180,E1 -24905.667,E2 -24905.667} C_VEL
LIN {X 0,Y 289.406,Z 579.166,A -85,B 0,C 180,E1 -24907.971,E2 -24907.971} C_VEL
LIN {X 0,Y 286.208,Z 587.22,A -85,B 0,C 180,E1 -24910.34,E2 -24910.34} C_VEL
LIN {X 0,Y 283.676,Z 593.753,A -85,B 0,C 180,E1 -24912.768,E2 -24912.768} C_VEL
LIN {X 0,Y 281.394,Z 599.601,A -85,B 0,C 180,E1 -24915.59,E2 -24915.59} C_VEL
LIN {X 0,Y 279.834,Z 603.927,A -85,B 0,C 180,E1 -24918.452,E2 -24918.452} C_VEL
LIN {X 0,Y 278.828,Z 606.846,A -85,B 0,C 180,E1 -24921.335,E2 -24921.335} C_VEL
LIN {X 0,Y 278.589,Z 608.442,A -85,B 0,C 180,E1 -24924.232,E2 -24924.232} C_VEL
LIN {X 0,Y 278.95,Z 608.814,A -85,B 0,C 180,E1 -24927.125,E2 -24927.125} C_VEL
LIN {X 0,Y 278.901,Z 613.084,A -85,B 0,C 180,E1 -24929.284,E2 -24929.284} C_VEL
LIN {X 0,Y 278.748,Z 616.401,A -85,B 0,C 180,E1 -24931.443,E2 -24931.443} C_VEL
LIN {X 0,Y 278.552,Z 619.411,A -85,B 0,C 180,E1 -24934.33,E2 -24934.33} C_VEL
LIN {X 0,Y 278.746,Z 621.033,A -85,B 0,C 180,E1 -24937.221,E2 -24937.221} C_VEL
LIN {X 0,Y 279.7,Z 621.333,A -85,B 0,C 180,E1 -24940.099,E2 -24940.099} C_VEL
LIN {X 0,Y 281.385,Z 620.316,A -85,B 0,C 180,E1 -24942.949,E2 -24942.949} C_VEL
LIN {X 0,Y 283.777,Z 617.981,A -85,B 0,C 180,E1 -24945.758,E2 -24945.758} C_VEL
LIN {X 0,Y 286.897,Z 614.293,A -85,B 0,C 180,E1 -24948.508,E2 -24948.508} C_VEL
LIN {X 0,Y 290.929,Z 609.151,A -85,B 0,C 180,E1 -24951.174,E2 -24951.174} C_VEL
LIN {X 0,Y 295.45,Z 602.478,A -85,B 0,C 180,E1 -24953.771,E2 -24953.771} C_VEL
LIN {X 0,Y 300.095,Z 595.153,A -85,B 0,C 180,E1 -24955.956,E2 -24955.956} C_VEL
LIN {X 0,Y 305.382,Z 586.197,A -85,B 0,C 180,E1 -24958.051,E2 -24958.051} C_VEL
LIN {X 0,Y 310.187,Z 577.054,A -85,B 0,C 180,E1 -24959.791,E2 -24959.791} C_VEL
LIN {X 0,Y 315.524,Z 566.119,A -85,B 0,C 180,E1 -24961.448,E2 -24961.448} C_VEL
LIN {X 0,Y 320.708,Z 554.133,A -85,B 0,C 180,E1 -24962.91,E2 -24962.91} C_VEL
LIN {X 0,Y 325.204,Z 542.381,A -85,B 0,C 180,E1 -24964.059,E2 -24964.059} C_VEL
LIN {X 0,Y 329.988,Z 527.924,A -85,B 0,C 180,E1 -24965.156,E2 -24965.156} C_VEL
LIN {X 0,Y 333.918,Z 513.682,A -85,B 0,C 180,E1 -24965.972,E2 -24965.972} C_VEL
LIN {X 0,Y 337.119,Z 498.652,A -85,B 0,C 180,E1 -24966.637,E2 -24966.637} C_VEL
LIN {X 0,Y 347.814,Z 428.371,A -85,B 0,C 180,E1 -24968.993,E2 -24968.993} C_VEL
LIN {X 0,Y 348.627,Z 414.553,A -85,B 0,C 180,E1 -24969.984,E2 -24969.984} C_VEL
LIN {X 0,Y 348.39,Z 413.598,A -85,B 0,C 180,E1 -24970.182,E2 -24970.182} C_VEL
LIN {X 0,Y 345.407,Z 407.997,A -85,B 0,C 180,E1 -24972.226,E2 -24972.226} C_VEL
LIN {X 0,Y 342.932,Z 403.75,A -85,B 0,C 180,E1 -24974.366,E2 -24974.366} C_VEL
LIN {X 0,Y 341.197,Z 401.173,A -85,B 0,C 180,E1 -24976.337,E2 -24976.337} C_VEL
LIN {X 0,Y 339.928,Z 399.07,A -85,B 0,C 180,E1 -24978.747,E2 -24978.747} C_VEL
LIN {X 0,Y 339.529,Z 398.691,A -85,B 0,C 180,E1 -24980.243,E2 -24980.243} C_VEL
LIN {X 0,Y 339.492,Z 399.313,A -85,B 0,C 180,E1 -24982.556,E2 -24982.556} C_VEL
LIN {X 0,Y 340.265,Z 401.392,A -85,B 0,C 180,E1 -24984.955,E2 -24984.955} C_VEL
LIN {X 0,Y 341.695,Z 404.431,A -85,B 0,C 180,E1 -24987.099,E2 -24987.099} C_VEL
LIN {X 0,Y 343.49,Z 408.531,A -85,B 0,C 180,E1 -24989.038,E2 -24989.038} C_VEL
LIN {X 0,Y 345.35,Z 413.087,A -85,B 0,C 180,E1 -24990.646,E2 -24990.646} C_VEL
LIN {X 0,Y 347.183,Z 417.736,A -85,B 0,C 180,E1 -24992.004,E2 -24992.004} C_VEL
LIN {X 0,Y 348.748,Z 422.526,A -85,B 0,C 180,E1 -24993.106,E2 -24993.106} C_VEL
LIN {X 0,Y 337.922,Z 492.892,A -85,B 0,C 180,E1 -24995.427,E2 -24995.427} C_VEL
LIN {X 0,Y 334.622,Z 508.364,A -85,B 0,C 180,E1 -24996.155,E2 -24996.155} C_VEL
LIN {X 0,Y 331.219,Z 521.24,A -85,B 0,C 180,E1 -24996.969,E2 -24996.969} C_VEL
LIN {X 0,Y 327.11,Z 534.131,A -85,B 0,C 180,E1 -24997.992,E2 -24997.992} C_VEL
LIN {X 0,Y 322.357,Z 546.934,A -85,B 0,C 180,E1 -24999.27,E2 -24999.27} C_VEL
LIN {X 0,Y 317.562,Z 558.153,A -85,B 0,C 180,E1 -25000.679,E2 -25000.679} C_VEL
LIN {X 0,Y 312.256,Z 569.112,A -85,B 0,C 180,E1 -25002.372,E2 -25002.372} C_VEL
LIN {X 0,Y 307.412,Z 578.201,A -85,B 0,C 180,E1 -25004.132,E2 -25004.132} C_VEL
LIN {X 0,Y 302.232,Z 587.003,A -85,B 0,C 180,E1 -25006.258,E2 -25006.258} C_VEL
LIN {X 0,Y 297.494,Z 594.217,A -85,B 0,C 180,E1 -25008.455,E2 -25008.455} C_VEL
LIN {X 0,Y 292.61,Z 600.721,A -85,B 0,C 180,E1 -25011.049,E2 -25011.049} C_VEL
LIN {X 0,Y 289.249,Z 604.751,A -85,B 0,C 180,E1 -25013.167,E2 -25013.167} C_VEL
LIN {X 0,Y 285.855,Z 608.307,A -85,B 0,C 180,E1 -25015.784,E2 -25015.784} C_VEL
LIN {X 0,Y 282.98,Z 610.633,A -85,B 0,C 180,E1 -25018.582,E2 -25018.582} C_VEL
LIN {X 0,Y 280.992,Z 611.605,A -85,B 0,C 180,E1 -25021.428,E2 -25021.428} C_VEL
LIN {X 0,Y 279.57,Z 611.242,A -85,B 0,C 180,E1 -25024.311,E2 -25024.311} C_VEL
LIN {X 0,Y 278.602,Z 609.508,A -85,B 0,C 180,E1 -25027.222,E2 -25027.222} C_VEL
LIN {X 0,Y 278.324,Z 606.364,A -85,B 0,C 180,E1 -25030.146,E2 -25030.146} C_VEL
LIN {X 0,Y 278.216,Z 602.974,A -85,B 0,C 180,E1 -25032.357,E2 -25032.357} C_VEL
LIN {X 0,Y 278.346,Z 598.644,A -85,B 0,C 180,E1 -25034.575,E2 -25034.575} C_VEL
LIN {X 0,Y 278.67,Z 592.02,A -85,B 0,C 180,E1 -25037.218,E2 -25037.218} C_VEL
LIN {X 0,Y 279.102,Z 583.858,A -85,B 0,C 180,E1 -25039.804,E2 -25039.804} C_VEL
LIN {X 0,Y 279.664,Z 575.096,A -85,B 0,C 180,E1 -25042.067,E2 -25042.067} C_VEL
LIN {X 0,Y 280.461,Z 564.396,A -85,B 0,C 180,E1 -25044.336,E2 -25044.336} C_VEL
LIN {X 0,Y 281.315,Z 553.835,A -85,B 0,C 180,E1 -25046.179,E2 -25046.179} C_VEL
LIN {X 0,Y 282.341,Z 541.795,A -85,B 0,C 180,E1 -25047.921,E2 -25047.921} C_VEL
LIN {X 0,Y 283.349,Z 529.114,A -85,B 0,C 180,E1 -25049.427,E2 -25049.427} C_VEL
LIN {X 0,Y 284.301,Z 516.349,A -85,B 0,C 180,E1 -25050.655,E2 -25050.655} C_VEL
LIN {X 0,Y 285.35,Z 501.786,A -85,B 0,C 180,E1 -25051.751,E2 -25051.751} C_VEL
LIN {X 0,Y 286.24,Z 486.687,A -85,B 0,C 180,E1 -25052.572,E2 -25052.572} C_VEL
LIN {X 0,Y 290.117,Z 387.677,A -85,B 0,C 180,E1 -25056.268,E2 -25056.268} C_VEL
LIN {X 0,Y 287.033,Z 356.83,A -85,B 0,C 180,E1 -25057.56,E2 -25057.56} C_VEL
LIN {X 0,Y 286.359,Z 346.613,A -85,B 0,C 180,E1 -25057.99,E2 -25057.99} C_VEL
LIN {X 0,Y 283.076,Z 330.143,A -85,B 0,C 180,E1 -25061.535,E2 -25061.535} C_VEL
LIN {X 0,Y 281.441,Z 321.986,A -85,B 0,C 180,E1 -25063.345,E2 -25063.345} C_VEL
LIN {X 0,Y 281.351,Z 321.995,A -85,B 0,C 180,E1 -25067.76,E2 -25067.76} C_VEL
LIN {X 0,Y 281.335,Z 321.996,A -85,B 0,C 180,E1 -25071.503,E2 -25071.503} C_VEL
LIN {X 0,Y 281.382,Z 321.979,A -85,B 0,C 180,E1 -25075.232,E2 -25075.232} C_VEL
LIN {X 0,Y 281.381,Z 321.993,A -85,B 0,C 180,E1 -25078.479,E2 -25078.479} C_VEL
LIN {X 0,Y 281.411,Z 321.978,A -85,B 0,C 180,E1 -25081.773,E2 -25081.773} C_VEL
LIN {X 0,Y 281.404,Z 321.989,A -85,B 0,C 180,E1 -25084.963,E2 -25084.963} C_VEL
LIN {X 0,Y 281.455,Z 321.984,A -85,B 0,C 180,E1 -25088.078,E2 -25088.078} C_VEL
LIN {X 0,Y 281.585,Z 322.049,A -85,B 0,C 180,E1 -25091.634,E2 -25091.634} C_VEL
LIN {X 0,Y 282.55,Z 324.754,A -85,B 0,C 180,E1 -25091.806,E2 -25091.806} C_VEL
LIN {X 0,Y 291.745,Z 344.76,A -85,B 0,C 180,E1 -25093.214,E2 -25093.214} C_VEL
LIN {X 0,Y 295.697,Z 354.805,A -85,B 0,C 180,E1 -25093.826,E2 -25093.826} C_VEL
LIN {X 0,Y 297.223,Z 359.957,A -85,B 0,C 180,E1 -25094.091,E2 -25094.091} C_VEL
LIN {X 0,Y 294.332,Z 451.614,A -85,B 0,C 180,E1 -25096.273,E2 -25096.273} C_VEL
LIN {X 0,Y 293.477,Z 466.159,A -85,B 0,C 180,E1 -25096.892,E2 -25096.892} C_VEL
LIN {X 0,Y 292.432,Z 479.469,A -85,B 0,C 180,E1 -25097.723,E2 -25097.723} C_VEL
LIN {X 0,Y 290.98,Z 493.385,A -85,B 0,C 180,E1 -25098.894,E2 -25098.894} C_VEL
LIN {X 0,Y 289.225,Z 505.886,A -85,B 0,C 180,E1 -25100.236,E2 -25100.236} C_VEL
LIN {X 0,Y 287.403,Z 517.302,A -85,B 0,C 180,E1 -25101.765,E2 -25101.765} C_VEL
LIN {X 0,Y 285.72,Z 528.698,A -85,B 0,C 180,E1 -25103.663,E2 -25103.663} C_VEL
LIN {X 0,Y 283.842,Z 538.946,A -85,B 0,C 180,E1 -25105.751,E2 -25105.751} C_VEL
LIN {X 0,Y 282.447,Z 547.395,A -85,B 0,C 180,E1 -25107.865,E2 -25107.865} C_VEL
LIN {X 0,Y 281.122,Z 554.457,A -85,B 0,C 180,E1 -25109.997,E2 -25109.997} C_VEL
LIN {X 0,Y 280.417,Z 560.837,A -85,B 0,C 180,E1 -25112.369,E2 -25112.369} C_VEL
LIN {X 0,Y 279.565,Z 566.542,A -85,B 0,C 180,E1 -25115.027,E2 -25115.027} C_VEL
LIN {X 0,Y 279.051,Z 570.135,A -85,B 0,C 180,E1 -25117.206,E2 -25117.206} C_VEL
LIN {X 0,Y 278.789,Z 573.665,A -85,B 0,C 180,E1 -25120.126,E2 -25120.126} C_VEL
LIN {X 0,Y 278.843,Z 575.805,A -85,B 0,C 180,E1 -25123.062,E2 -25123.062} C_VEL
LIN {X 0,Y 279.256,Z 576.587,A -85,B 0,C 180,E1 -25126.012,E2 -25126.012} C_VEL
LIN {X 0,Y 280.129,Z 575.99,A -85,B 0,C 180,E1 -25128.965,E2 -25128.965} C_VEL
LIN {X 0,Y 281.461,Z 573.999,A -85,B 0,C 180,E1 -25131.915,E2 -25131.915} C_VEL
LIN {X 0,Y 283.413,Z 570.552,A -85,B 0,C 180,E1 -25134.84,E2 -25134.84} C_VEL
LIN {X 0,Y 285.92,Z 565.535,A -85,B 0,C 180,E1 -25137.736,E2 -25137.736} C_VEL
LIN {X 0,Y 288.216,Z 560.619,A -85,B 0,C 180,E1 -25139.877,E2 -25139.877} C_VEL
LIN {X 0,Y 290.852,Z 554.606,A -85,B 0,C 180,E1 -25141.988,E2 -25141.988} C_VEL
LIN {X 0,Y 293.765,Z 547.303,A -85,B 0,C 180,E1 -25144.074,E2 -25144.074} C_VEL
LIN {X 0,Y 297.058,Z 538.441,A -85,B 0,C 180,E1 -25146.116,E2 -25146.116} C_VEL
LIN {X 0,Y 300.095,Z 529.617,A -85,B 0,C 180,E1 -25147.78,E2 -25147.78} C_VEL
LIN {X 0,Y 303.297,Z 519.009,A -85,B 0,C 180,E1 -25149.422,E2 -25149.422} C_VEL
LIN {X 0,Y 306.423,Z 507.09,A -85,B 0,C 180,E1 -25150.908,E2 -25150.908} C_VEL
LIN {X 0,Y 309.176,Z 494.552,A -85,B 0,C 180,E1 -25152.152,E2 -25152.152} C_VEL
LIN {X 0,Y 311.383,Z 481.145,A -85,B 0,C 180,E1 -25153.205,E2 -25153.205} C_VEL
LIN {X 0,Y 313.279,Z 466.862,A -85,B 0,C 180,E1 -25154.019,E2 -25154.019} C_VEL
LIN {X 0,Y 314.5,Z 453.072,A -85,B 0,C 180,E1 -25154.557,E2 -25154.557} C_VEL
LIN {X 0,Y 317.817,Z 383.145,A -85,B 0,C 180,E1 -25156.127,E2 -25156.127} C_VEL
LIN {X 0,Y 310.14,Z 367.135,A -85,B 0,C 180,E1 -25157.786,E2 -25157.786} C_VEL
LIN {X 0,Y 305.066,Z 357.956,A -85,B 0,C 180,E1 -25158.91,E2 -25158.91} C_VEL
LIN {X 0,Y 296.001,Z 343.69,A -85,B 0,C 180,E1 -25161.001,E2 -25161.001} C_VEL
LIN {X 0,Y 289.99,Z 335.076,A -85,B 0,C 180,E1 -25162.48,E2 -25162.48} C_VEL
LIN {X 0,Y 287.223,Z 331.1,A -85,B 0,C 180,E1 -25163.196,E2 -25163.196} C_VEL
LIN {X 0,Y 284.849,Z 327.614,A -85,B 0,C 180,E1 -25163.832,E2 -25163.832} C_VEL
LIN {X 0,Y 284.05,Z 326.667,A -85,B 0,C 180,E1 -25164.042,E2 -25164.042} C_VEL
LIN {X 0,Y 282.195,Z 324.493,A -85,B 0,C 180,E1 -25164.536,E2 -25164.536} C_VEL
LIN {X 0,Y 281.354,Z 321.957,A -85,B 0,C 180,E1 -25164.851,E2 -25164.851} C_VEL
LIN {X 0,Y 281.375,Z 321.985,A -85,B 0,C 180,E1 -25168.482,E2 -25168.482} C_VEL
LIN {X 0,Y 281.399,Z 321.982,A -85,B 0,C 180,E1 -25171.775,E2 -25171.775} C_VEL
LIN {X 0,Y 281.427,Z 321.988,A -85,B 0,C 180,E1 -25174.969,E2 -25174.969} C_VEL
LIN {X 0,Y 281.43,Z 321.98,A -85,B 0,C 180,E1 -25178.079,E2 -25178.079} C_VEL
LIN {X 0,Y 281.485,Z 321.963,A -85,B 0,C 180,E1 -25181.126,E2 -25181.126} C_VEL
LIN {X 0,Y 281.614,Z 321.944,A -85,B 0,C 180,E1 -25185.919,E2 -25185.919} C_VEL
LIN {X 0,Y 281.661,Z 321.943,A -85,B 0,C 180,E1 -25189.975,E2 -25189.975} C_VEL
LIN {X 0,Y 281.849,Z 321.934,A -85,B 0,C 180,E1 -25194.295,E2 -25194.295} C_VEL
LIN {X 0,Y 281.9,Z 321.908,A -85,B 0,C 180,E1 -25197.152,E2 -25197.152} C_VEL
LIN {X 0,Y 281.973,Z 321.901,A -85,B 0,C 180,E1 -25200.79,E2 -25200.79} C_VEL
LIN {X 0,Y 281.923,Z 321.923,A -85,B 0,C 180,E1 -25204.275,E2 -25204.275} C_VEL
LIN {X 0,Y 281.809,Z 321.916,A -85,B 0,C 180,E1 -25206.981,E2 -25206.981} C_VEL
LIN {X 0,Y 281.07,Z 322.012,A -85,B 0,C 180,E1 -25208.172,E2 -25208.172} C_VEL
LIN {X 0,Y 278.176,Z 322.389,A -85,B 0,C 180,E1 -25210.111,E2 -25210.111} C_VEL
LIN {X 0,Y 275.751,Z 322.678,A -85,B 0,C 180,E1 -25211.685,E2 -25211.685} C_VEL
LIN {X 0,Y 274.697,Z 322.802,A -85,B 0,C 180,E1 -25212.906,E2 -25212.906} C_VEL
LIN {X 0,Y 274.602,Z 322.815,A -85,B 0,C 180,E1 -25213.32,E2 -25213.32} C_VEL
LIN {X 0,Y 274.437,Z 322.835,A -85,B 0,C 180,E1 -25217.835,E2 -25217.835} C_VEL
LIN {X 0,Y 274.391,Z 322.852,A -85,B 0,C 180,E1 -25220.94,E2 -25220.94} C_VEL
LIN {X 0,Y 274.361,Z 322.865,A -85,B 0,C 180,E1 -25224.109,E2 -25224.109} C_VEL
LIN {X 0,Y 274.342,Z 322.858,A -85,B 0,C 180,E1 -25227.36,E2 -25227.36} C_VEL
LIN {X 0,Y 274.318,Z 322.86,A -85,B 0,C 180,E1 -25230.709,E2 -25230.709} C_VEL
LIN {X 0,Y 274.348,Z 322.833,A -85,B 0,C 180,E1 -25234.173,E2 -25234.173} C_VEL
LIN {X 0,Y 274.382,Z 322.862,A -85,B 0,C 180,E1 -25237.899,E2 -25237.899} C_VEL
LIN {X 0,Y 276.745,Z 330.387,A -85,B 0,C 180,E1 -25241.824,E2 -25241.824} C_VEL
LIN {X 0,Y 279.002,Z 337.854,A -85,B 0,C 180,E1 -25245.342,E2 -25245.342} C_VEL
LIN {X 0,Y 280.082,Z 341.53,A -85,B 0,C 180,E1 -25246.878,E2 -25246.878} C_VEL
LIN {X 0,Y 282.467,Z 345.757,A -85,B 0,C 180,E1 -25247.565,E2 -25247.565} C_VEL
LIN {X 0,Y 283.949,Z 348.063,A -85,B 0,C 180,E1 -25247.971,E2 -25247.971} C_VEL
LIN {X 0,Y 290.219,Z 358.883,A -85,B 0,C 180,E1 -25249.646,E2 -25249.646} C_VEL
LIN {X 0,Y 297.428,Z 372.663,A -85,B 0,C 180,E1 -25251.472,E2 -25251.472} C_VEL
LIN {X 0,Y 304.328,Z 387.569,A -85,B 0,C 180,E1 -25253.14,E2 -25253.14} C_VEL
LIN {X 0,Y 306.565,Z 393.334,A -85,B 0,C 180,E1 -25253.685,E2 -25253.685} C_VEL
LIN {X 0,Y 309.586,Z 415.111,A -85,B 0,C 180,E1 -25254.819,E2 -25254.819} C_VEL
LIN {X 0,Y 310.526,Z 423.883,A -85,B 0,C 180,E1 -25255.223,E2 -25255.223} C_VEL
LIN {X 0,Y 307.59,Z 481.881,A -85,B 0,C 180,E1 -25256.535,E2 -25256.535} C_VEL
LIN {X 0,Y 306.059,Z 496.322,A -85,B 0,C 180,E1 -25257.079,E2 -25257.079} C_VEL
LIN {X 0,Y 303.63,Z 510.801,A -85,B 0,C 180,E1 -25257.862,E2 -25257.862} C_VEL
LIN {X 0,Y 300.839,Z 523.65,A -85,B 0,C 180,E1 -25258.803,E2 -25258.803} C_VEL
LIN {X 0,Y 297.676,Z 536.138,A -85,B 0,C 180,E1 -25260.003,E2 -25260.003} C_VEL
LIN {X 0,Y 294.23,Z 547.564,A -85,B 0,C 180,E1 -25261.378,E2 -25261.378} C_VEL
LIN {X 0,Y 290.48,Z 559.342,A -85,B 0,C 180,E1 -25263.183,E2 -25263.183} C_VEL
LIN {X 0,Y 286.752,Z 569.36,A -85,B 0,C 180,E1 -25265.084,E2 -25265.084} C_VEL
LIN {X 0,Y 283.37,Z 577.906,A -85,B 0,C 180,E1 -25267.092,E2 -25267.092} C_VEL
LIN {X 0,Y 279.934,Z 586.131,A -85,B 0,C 180,E1 -25269.498,E2 -25269.498} C_VEL
LIN {X 0,Y 277.564,Z 591.916,A -85,B 0,C 180,E1 -25271.616,E2 -25271.616} C_VEL
LIN {X 0,Y 275.041,Z 598.129,A -85,B 0,C 180,E1 -25274.494,E2 -25274.494} C_VEL
LIN {X 0,Y 273.567,Z 601.709,A -85,B 0,C 180,E1 -25276.681,E2 -25276.681} C_VEL
LIN {X 0,Y 272.202,Z 605.26,A -85,B 0,C 180,E1 -25279.627,E2 -25279.627} C_VEL
LIN {X 0,Y 271.506,Z 607.454,A -85,B 0,C 180,E1 -25282.592,E2 -25282.592} C_VEL
LIN {X 0,Y 271.618,Z 608.352,A -85,B 0,C 180,E1 -25285.567,E2 -25285.567} C_VEL
LIN {X 0,Y 271.905,Z 608.454,A -85,B 0,C 180,E1 -25287.42,E2 -25287.42} C_VEL
LIN {X 0,Y 271.816,Z 613.353,A -85,B 0,C 180,E1 -25290.004,E2 -25290.004} C_VEL
LIN {X 0,Y 271.718,Z 615.565,A -85,B 0,C 180,E1 -25291.481,E2 -25291.481} C_VEL
LIN {X 0,Y 271.492,Z 618.818,A -85,B 0,C 180,E1 -25294.443,E2 -25294.443} C_VEL
LIN {X 0,Y 271.69,Z 620.672,A -85,B 0,C 180,E1 -25297.41,E2 -25297.41} C_VEL
LIN {X 0,Y 272.698,Z 621.206,A -85,B 0,C 180,E1 -25300.362,E2 -25300.362} C_VEL
LIN {X 0,Y 274.48,Z 620.43,A -85,B 0,C 180,E1 -25303.281,E2 -25303.281} C_VEL
LIN {X 0,Y 276.954,Z 618.352,A -85,B 0,C 180,E1 -25306.156,E2 -25306.156} C_VEL
LIN {X 0,Y 280.2,Z 614.939,A -85,B 0,C 180,E1 -25308.967,E2 -25308.967} C_VEL
LIN {X 0,Y 284.384,Z 610.076,A -85,B 0,C 180,E1 -25311.685,E2 -25311.685} C_VEL
LIN {X 0,Y 289.066,Z 603.717,A -85,B 0,C 180,E1 -25314.33,E2 -25314.33} C_VEL
LIN {X 0,Y 293.887,Z 596.752,A -85,B 0,C 180,E1 -25316.547,E2 -25316.547} C_VEL
LIN {X 0,Y 299.32,Z 588.239,A -85,B 0,C 180,E1 -25318.671,E2 -25318.671} C_VEL
LIN {X 0,Y 304.29,Z 579.548,A -85,B 0,C 180,E1 -25320.429,E2 -25320.429} C_VEL
LIN {X 0,Y 309.754,Z 569.221,A -85,B 0,C 180,E1 -25322.103,E2 -25322.103} C_VEL
LIN {X 0,Y 315.075,Z 557.935,A -85,B 0,C 180,E1 -25323.576,E2 -25323.576} C_VEL
LIN {X 0,Y 320.179,Z 545.653,A -85,B 0,C 180,E1 -25324.86,E2 -25324.86} C_VEL
LIN {X 0,Y 325.079,Z 532.08,A -85,B 0,C 180,E1 -25325.958,E2 -25325.958} C_VEL
LIN {X 0,Y 329.364,Z 518.1,A -85,B 0,C 180,E1 -25326.834,E2 -25326.834} C_VEL
LIN {X 0,Y 333.169,Z 502.354,A -85,B 0,C 180,E1 -25327.57,E2 -25327.57} C_VEL
LIN {X 0,Y 337.017,Z 479.378,A -85,B 0,C 180,E1 -25328.386,E2 -25328.386} C_VEL
LIN {X 0,Y 344.827,Z 430.042,A -85,B 0,C 180,E1 -25330.03,E2 -25330.03} C_VEL
LIN {X 0,Y 345.613,Z 419.068,A -85,B 0,C 180,E1 -25330.833,E2 -25330.833} C_VEL
LIN {X 0,Y 343.178,Z 414.278,A -85,B 0,C 180,E1 -25332.647,E2 -25332.647} C_VEL
LIN {X 0,Y 341.082,Z 410.501,A -85,B 0,C 180,E1 -25334.57,E2 -25334.57} C_VEL
LIN {X 0,Y 339.294,Z 407.671,A -85,B 0,C 180,E1 -25336.789,E2 -25336.789} C_VEL
LIN {X 0,Y 338.331,Z 405.977,A -85,B 0,C 180,E1 -25338.789,E2 -25338.789} C_VEL
LIN {X 0,Y 337.978,Z 405.611,A -85,B 0,C 180,E1 -25340.072,E2 -25340.072} C_VEL
LIN {X 0,Y 337.881,Z 406.145,A -85,B 0,C 180,E1 -25342.346,E2 -25342.346} C_VEL
LIN {X 0,Y 338.574,Z 408.17,A -85,B 0,C 180,E1 -25344.754,E2 -25344.754} C_VEL
LIN {X 0,Y 339.798,Z 410.944,A -85,B 0,C 180,E1 -25346.759,E2 -25346.759} C_VEL
LIN {X 0,Y 341.492,Z 415.151,A -85,B 0,C 180,E1 -25348.758,E2 -25348.758} C_VEL
LIN {X 0,Y 343.304,Z 419.896,A -85,B 0,C 180,E1 -25350.423,E2 -25350.423} C_VEL
LIN {X 0,Y 345.248,Z 425.568,A -85,B 0,C 180,E1 -25351.972,E2 -25351.972} C_VEL
LIN {X 0,Y 345.455,Z 426.166,A -85,B 0,C 180,E1 -25352.123,E2 -25352.123} C_VEL
LIN {X 0,Y 334.586,Z 493.729,A -85,B 0,C 180,E1 -25354.37,E2 -25354.37} C_VEL
LIN {X 0,Y 331.299,Z 508.511,A -85,B 0,C 180,E1 -25355.069,E2 -25355.069} C_VEL
LIN {X 0,Y 327.729,Z 521.379,A -85,B 0,C 180,E1 -25355.873,E2 -25355.873} C_VEL
LIN {X 0,Y 322.935,Z 535.727,A -85,B 0,C 180,E1 -25357.019,E2 -25357.019} C_VEL
LIN {X 0,Y 318.006,Z 548.163,A -85,B 0,C 180,E1 -25358.295,E2 -25358.295} C_VEL
LIN {X 0,Y 312.664,Z 559.918,A -85,B 0,C 180,E1 -25359.801,E2 -25359.801} C_VEL
LIN {X 0,Y 307.475,Z 570.005,A -85,B 0,C 180,E1 -25361.402,E2 -25361.402} C_VEL
LIN {X 0,Y 302.372,Z 578.994,A -85,B 0,C 180,E1 -25363.168,E2 -25363.168} C_VEL
LIN {X 0,Y 296.829,Z 587.852,A -85,B 0,C 180,E1 -25365.362,E2 -25365.362} C_VEL
LIN {X 0,Y 291.943,Z 594.761,A -85,B 0,C 180,E1 -25367.53,E2 -25367.53} C_VEL
LIN {X 0,Y 286.819,Z 601.159,A -85,B 0,C 180,E1 -25370.157,E2 -25370.157} C_VEL
LIN {X 0,Y 282.37,Z 605.969,A -85,B 0,C 180,E1 -25372.875,E2 -25372.875} C_VEL
LIN {X 0,Y 278.737,Z 609.295,A -85,B 0,C 180,E1 -25375.676,E2 -25375.676} C_VEL
LIN {X 0,Y 275.848,Z 611.24,A -85,B 0,C 180,E1 -25378.545,E2 -25378.545} C_VEL
LIN {X 0,Y 273.843,Z 611.839,A -85,B 0,C 180,E1 -25381.466,E2 -25381.466} C_VEL
LIN {X 0,Y 272.392,Z 611.111,A -85,B 0,C 180,E1 -25384.424,E2 -25384.424} C_VEL
LIN {X 0,Y 271.47,Z 609.005,A -85,B 0,C 180,E1 -25387.412,E2 -25387.412} C_VEL
LIN {X 0,Y 271.258,Z 605.46,A -85,B 0,C 180,E1 -25390.414,E2 -25390.414} C_VEL
LIN {X 0,Y 271.155,Z 601.76,A -85,B 0,C 180,E1 -25392.684,E2 -25392.684} C_VEL
LIN {X 0,Y 271.328,Z 597.034,A -85,B 0,C 180,E1 -25394.96,E2 -25394.96} C_VEL
LIN {X 0,Y 271.615,Z 590.751,A -85,B 0,C 180,E1 -25397.406,E2 -25397.406} C_VEL
LIN {X 0,Y 272.066,Z 582.682,A -85,B 0,C 180,E1 -25399.946,E2 -25399.946} C_VEL
LIN {X 0,Y 272.626,Z 574.014,A -85,B 0,C 180,E1 -25402.177,E2 -25402.177} C_VEL
LIN {X 0,Y 273.431,Z 563.563,A -85,B 0,C 180,E1 -25404.398,E2 -25404.398} C_VEL
LIN {X 0,Y 274.317,Z 552.705,A -85,B 0,C 180,E1 -25406.312,E2 -25406.312} C_VEL
LIN {X 0,Y 275.317,Z 540.62,A -85,B 0,C 180,E1 -25408.077,E2 -25408.077} C_VEL
LIN {X 0,Y 276.352,Z 527.68,A -85,B 0,C 180,E1 -25409.62,E2 -25409.62} C_VEL
LIN {X 0,Y 277.389,Z 514.057,A -85,B 0,C 180,E1 -25410.917,E2 -25410.917} C_VEL
LIN {X 0,Y 278.388,Z 499.195,A -85,B 0,C 180,E1 -25412.002,E2 -25412.002} C_VEL
LIN {X 0,Y 279.274,Z 484.305,A -85,B 0,C 180,E1 -25412.792,E2 -25412.792} C_VEL
LIN {X 0,Y 283.1,Z 387.906,A -85,B 0,C 180,E1 -25416.497,E2 -25416.497} C_VEL
LIN {X 0,Y 280.138,Z 358.049,A -85,B 0,C 180,E1 -25417.778,E2 -25417.778} C_VEL
LIN {X 0,Y 279.264,Z 347.246,A -85,B 0,C 180,E1 -25418.24,E2 -25418.24} C_VEL
LIN {X 0,Y 278.901,Z 345.333,A -85,B 0,C 180,E1 -25418.58,E2 -25418.58} C_VEL
LIN {X 0,Y 275.361,Z 327.665,A -85,B 0,C 180,E1 -25422.461,E2 -25422.461} C_VEL
LIN {X 0,Y 274.368,Z 322.867,A -85,B 0,C 180,E1 -25423.574,E2 -25423.574} C_VEL
LIN {X 0,Y 274.329,Z 322.872,A -85,B 0,C 180,E1 -25428.401,E2 -25428.401} C_VEL
LIN {X 0,Y 274.318,Z 322.874,A -85,B 0,C 180,E1 -25432.331,E2 -25432.331} C_VEL
LIN {X 0,Y 274.333,Z 322.853,A -85,B 0,C 180,E1 -25435.822,E2 -25435.822} C_VEL
LIN {X 0,Y 274.307,Z 322.873,A -85,B 0,C 180,E1 -25439.286,E2 -25439.286} C_VEL
LIN {X 0,Y 274.38,Z 322.86,A -85,B 0,C 180,E1 -25443.315,E2 -25443.315} C_VEL
LIN {X 0,Y 274.413,Z 322.861,A -85,B 0,C 180,E1 -25447.484,E2 -25447.484} C_VEL
LIN {X 0,Y 274.496,Z 322.849,A -85,B 0,C 180,E1 -25450.928,E2 -25450.928} C_VEL
LIN {X 0,Y 275.628,Z 325.833,A -85,B 0,C 180,E1 -25451.139,E2 -25451.139} C_VEL
LIN {X 0,Y 284.996,Z 345.966,A -85,B 0,C 180,E1 -25452.628,E2 -25452.628} C_VEL
LIN {X 0,Y 289.602,Z 357.518,A -85,B 0,C 180,E1 -25453.365,E2 -25453.365} C_VEL
LIN {X 0,Y 290.721,Z 361.182,A -85,B 0,C 180,E1 -25453.562,E2 -25453.562} C_VEL
LIN {X 0,Y 287.745,Z 452.122,A -85,B 0,C 180,E1 -25455.773,E2 -25455.773} C_VEL
LIN {X 0,Y 286.845,Z 466.638,A -85,B 0,C 180,E1 -25456.403,E2 -25456.403} C_VEL
LIN {X 0,Y 285.77,Z 479.928,A -85,B 0,C 180,E1 -25457.253,E2 -25457.253} C_VEL
LIN {X 0,Y 284.279,Z 493.83,A -85,B 0,C 180,E1 -25458.448,E2 -25458.448} C_VEL
LIN {X 0,Y 282.468,Z 506.326,A -85,B 0,C 180,E1 -25459.82,E2 -25459.82} C_VEL
LIN {X 0,Y 280.59,Z 517.737,A -85,B 0,C 180,E1 -25461.382,E2 -25461.382} C_VEL
LIN {X 0,Y 278.987,Z 528.163,A -85,B 0,C 180,E1 -25463.147,E2 -25463.147} C_VEL
LIN {X 0,Y 277.081,Z 538.578,A -85,B 0,C 180,E1 -25465.284,E2 -25465.284} C_VEL
LIN {X 0,Y 275.573,Z 547.161,A -85,B 0,C 180,E1 -25467.447,E2 -25467.447} C_VEL
LIN {X 0,Y 274.037,Z 555.414,A -85,B 0,C 180,E1 -25469.996,E2 -25469.996} C_VEL
LIN {X 0,Y 273.375,Z 561.153,A -85,B 0,C 180,E1 -25472.203,E2 -25472.203} C_VEL
LIN {X 0,Y 272.653,Z 565.886,A -85,B 0,C 180,E1 -25474.416,E2 -25474.416} C_VEL
LIN {X 0,Y 271.923,Z 570.826,A -85,B 0,C 180,E1 -25477.396,E2 -25477.396} C_VEL
LIN {X 0,Y 271.705,Z 574.27,A -85,B 0,C 180,E1 -25480.393,E2 -25480.393} C_VEL
LIN {X 0,Y 271.788,Z 576.322,A -85,B 0,C 180,E1 -25483.408,E2 -25483.408} C_VEL
LIN {X 0,Y 272.277,Z 576.997,A -85,B 0,C 180,E1 -25486.434,E2 -25486.434} C_VEL
LIN {X 0,Y 273.229,Z 576.308,A -85,B 0,C 180,E1 -25489.463,E2 -25489.463} C_VEL
LIN {X 0,Y 274.689,Z 574.232,A -85,B 0,C 180,E1 -25492.484,E2 -25492.484} C_VEL
LIN {X 0,Y 276.768,Z 570.697,A -85,B 0,C 180,E1 -25495.478,E2 -25495.478} C_VEL
LIN {X 0,Y 279.412,Z 565.586,A -85,B 0,C 180,E1 -25498.44,E2 -25498.44} C_VEL
LIN {X 0,Y 281.872,Z 560.568,A -85,B 0,C 180,E1 -25500.621,E2 -25500.621} C_VEL
LIN {X 0,Y 284.644,Z 554.443,A -85,B 0,C 180,E1 -25502.772,E2 -25502.772} C_VEL
LIN {X 0,Y 287.718,Z 547.014,A -85,B 0,C 180,E1 -25504.892,E2 -25504.892} C_VEL
LIN {X 0,Y 291.164,Z 538.008,A -85,B 0,C 180,E1 -25506.967,E2 -25506.967} C_VEL
LIN {X 0,Y 294.329,Z 529.012,A -85,B 0,C 180,E1 -25508.655,E2 -25508.655} C_VEL
LIN {X 0,Y 297.667,Z 518.195,A -85,B 0,C 180,E1 -25510.319,E2 -25510.319} C_VEL
LIN {X 0,Y 301.026,Z 505.539,A -85,B 0,C 180,E1 -25511.876,E2 -25511.876} C_VEL
LIN {X 0,Y 303.724,Z 493.104,A -85,B 0,C 180,E1 -25513.09,E2 -25513.09} C_VEL
LIN {X 0,Y 306.09,Z 479.19,A -85,B 0,C 180,E1 -25514.143,E2 -25514.143} C_VEL
LIN {X 0,Y 307.93,Z 464.82,A -85,B 0,C 180,E1 -25514.919,E2 -25514.919} C_VEL
LIN {X 0,Y 309.044,Z 451.576,A -85,B 0,C 180,E1 -25515.405,E2 -25515.405} C_VEL
LIN {X 0,Y 312.23,Z 385.367,A -85,B 0,C 180,E1 -25516.908,E2 -25516.908} C_VEL
LIN {X 0,Y 304.86,Z 370.084,A -85,B 0,C 180,E1 -25518.565,E2 -25518.565} C_VEL
LIN {X 0,Y 300.241,Z 361.823,A -85,B 0,C 180,E1 -25519.626,E2 -25519.626} C_VEL
LIN {X 0,Y 292.112,Z 348.867,A -85,B 0,C 180,E1 -25521.576,E2 -25521.576} C_VEL
LIN {X 0,Y 285.988,Z 339.99,A -85,B 0,C 180,E1 -25523.137,E2 -25523.137} C_VEL
LIN {X 0,Y 283.379,Z 336.288,A -85,B 0,C 180,E1 -25523.834,E2 -25523.834} C_VEL
LIN {X 0,Y 280.656,Z 332.4,A -85,B 0,C 180,E1 -25524.586,E2 -25524.586} C_VEL
LIN {X 0,Y 278.361,Z 329.436,A -85,B 0,C 180,E1 -25525.23,E2 -25525.23} C_VEL
LIN {X 0,Y 277.511,Z 327.942,A -85,B 0,C 180,E1 -25525.489,E2 -25525.489} C_VEL
LIN {X 0,Y 275.392,Z 325.871,A -85,B 0,C 180,E1 -25526.083,E2 -25526.083} C_VEL
LIN {X 0,Y 274.394,Z 323.395,A -85,B 0,C 180,E1 -25526.429,E2 -25526.429} C_VEL
LIN {X 0,Y 274.302,Z 322.858,A -85,B 0,C 180,E1 -25526.524,E2 -25526.524} C_VEL
LIN {X 0,Y 274.327,Z 322.873,A -85,B 0,C 180,E1 -25530.979,E2 -25530.979} C_VEL
LIN {X 0,Y 274.358,Z 322.866,A -85,B 0,C 180,E1 -25534.277,E2 -25534.277} C_VEL
LIN {X 0,Y 274.39,Z 322.85,A -85,B 0,C 180,E1 -25537.486,E2 -25537.486} C_VEL
LIN {X 0,Y 274.442,Z 322.84,A -85,B 0,C 180,E1 -25540.778,E2 -25540.778} C_VEL
LIN {X 0,Y 274.555,Z 322.823,A -85,B 0,C 180,E1 -25545.784,E2 -25545.784} C_VEL
LIN {X 0,Y 274.6,Z 322.826,A -85,B 0,C 180,E1 -25549.714,E2 -25549.714} C_VEL
LIN {X 0,Y 274.819,Z 322.81,A -85,B 0,C 180,E1 -25554.149,E2 -25554.149} C_VEL
LIN {X 0,Y 274.941,Z 322.793,A -85,B 0,C 180,E1 -25558.54,E2 -25558.54} C_VEL
LIN {X 0,Y 274.941,Z 322.771,A -85,B 0,C 180,E1 -25561.46,E2 -25561.46} C_VEL
LIN {X 0,Y 274.82,Z 322.798,A -85,B 0,C 180,E1 -25565.852,E2 -25565.852} C_VEL
LIN {X 0,Y 274.631,Z 322.831,A -85,B 0,C 180,E1 -25570.284,E2 -25570.284} C_VEL
LIN {X 0,Y 274.602,Z 322.815,A -85,B 0,C 180,E1 -25573.32,E2 -25573.32} C_VEL
LIN {X 0,Y 273.902,Z 322.918,A -85,B 0,C 180,E1 -25574.542,E2 -25574.542} C_VEL
LIN {X 0,Y 271.011,Z 323.272,A -85,B 0,C 180,E1 -25576.531,E2 -25576.531} C_VEL
LIN {X 0,Y 268.557,Z 323.579,A -85,B 0,C 180,E1 -25578.148,E2 -25578.148} C_VEL
LIN {X 0,Y 267.486,Z 323.717,A -85,B 0,C 180,E1 -25579.402,E2 -25579.402} C_VEL
LIN {X 0,Y 267.387,Z 323.733,A -85,B 0,C 180,E1 -25579.828,E2 -25579.828} C_VEL
LIN {X 0,Y 267.336,Z 323.732,A -85,B 0,C 180,E1 -25583.515,E2 -25583.515} C_VEL
LIN {X 0,Y 267.304,Z 323.732,A -85,B 0,C 180,E1 -25587.019,E2 -25587.019} C_VEL
LIN {X 0,Y 267.275,Z 323.737,A -85,B 0,C 180,E1 -25590.146,E2 -25590.146} C_VEL
LIN {X 0,Y 267.301,Z 323.726,A -85,B 0,C 180,E1 -25593.387,E2 -25593.387} C_VEL
LIN {X 0,Y 267.322,Z 323.836,A -85,B 0,C 180,E1 -25596.304,E2 -25596.304} C_VEL
LIN {X 0,Y 269.223,Z 329.606,A -85,B 0,C 180,E1 -25599.6,E2 -25599.6} C_VEL
LIN {X 0,Y 271.802,Z 337.981,A -85,B 0,C 180,E1 -25603.822,E2 -25603.822} C_VEL
LIN {X 0,Y 272.629,Z 340.808,A -85,B 0,C 180,E1 -25605.084,E2 -25605.084} C_VEL
LIN {X 0,Y 275.46,Z 345.544,A -85,B 0,C 180,E1 -25605.961,E2 -25605.961} C_VEL
LIN {X 0,Y 276.905,Z 347.9,A -85,B 0,C 180,E1 -25606.393,E2 -25606.393} C_VEL
LIN {X 0,Y 280.565,Z 354.036,A -85,B 0,C 180,E1 -25607.455,E2 -25607.455} C_VEL
LIN {X 0,Y 285.96,Z 363.326,A -85,B 0,C 180,E1 -25608.943,E2 -25608.943} C_VEL
LIN {X 0,Y 292.955,Z 376.896,A -85,B 0,C 180,E1 -25610.789,E2 -25610.789} C_VEL
LIN {X 0,Y 300.198,Z 392.951,A -85,B 0,C 180,E1 -25612.612,E2 -25612.612} C_VEL
LIN {X 0,Y 301.474,Z 396.636,A -85,B 0,C 180,E1 -25612.946,E2 -25612.946} C_VEL
LIN {X 0,Y 304.342,Z 417.96,A -85,B 0,C 180,E1 -25614.081,E2 -25614.081} C_VEL
LIN {X 0,Y 305.015,Z 425.393,A -85,B 0,C 180,E1 -25614.415,E2 -25614.415} C_VEL
LIN {X 0,Y 301.983,Z 482.202,A -85,B 0,C 180,E1 -25615.721,E2 -25615.721} C_VEL
LIN {X 0,Y 300.387,Z 496.501,A -85,B 0,C 180,E1 -25616.276,E2 -25616.276} C_VEL
LIN {X 0,Y 297.899,Z 510.821,A -85,B 0,C 180,E1 -25617.066,E2 -25617.066} C_VEL
LIN {X 0,Y 294.833,Z 524.446,A -85,B 0,C 180,E1 -25618.094,E2 -25618.094} C_VEL
LIN {X 0,Y 291.581,Z 536.697,A -85,B 0,C 180,E1 -25619.309,E2 -25619.309} C_VEL
LIN {X 0,Y 287.69,Z 549.103,A -85,B 0,C 180,E1 -25620.865,E2 -25620.865} C_VEL
LIN {X 0,Y 284.075,Z 559.812,A -85,B 0,C 180,E1 -25622.58,E2 -25622.58} C_VEL
LIN {X 0,Y 280.342,Z 569.463,A -85,B 0,C 180,E1 -25624.473,E2 -25624.473} C_VEL
LIN {X 0,Y 276.848,Z 577.93,A -85,B 0,C 180,E1 -25626.521,E2 -25626.521} C_VEL
LIN {X 0,Y 273.276,Z 586.055,A -85,B 0,C 180,E1 -25628.975,E2 -25628.975} C_VEL
LIN {X 0,Y 270.803,Z 591.805,A -85,B 0,C 180,E1 -25631.14,E2 -25631.14} C_VEL
LIN {X 0,Y 268.169,Z 597.924,A -85,B 0,C 180,E1 -25634.086,E2 -25634.086} C_VEL
LIN {X 0,Y 266.535,Z 601.713,A -85,B 0,C 180,E1 -25636.494,E2 -25636.494} C_VEL
LIN {X 0,Y 265.193,Z 604.966,A -85,B 0,C 180,E1 -25639.349,E2 -25639.349} C_VEL
LIN {X 0,Y 264.444,Z 607.106,A -85,B 0,C 180,E1 -25642.393,E2 -25642.393} C_VEL
LIN {X 0,Y 264.537,Z 607.95,A -85,B 0,C 180,E1 -25645.448,E2 -25645.448} C_VEL
LIN {X 0,Y 264.904,Z 607.849,A -85,B 0,C 180,E1 -25647.636,E2 -25647.636} C_VEL
LIN {X 0,Y 264.791,Z 612.378,A -85,B 0,C 180,E1 -25650.004,E2 -25650.004} C_VEL
LIN {X 0,Y 264.692,Z 614.691,A -85,B 0,C 180,E1 -25651.52,E2 -25651.52} C_VEL
LIN {X 0,Y 264.439,Z 618.156,A -85,B 0,C 180,E1 -25654.561,E2 -25654.561} C_VEL
LIN {X 0,Y 264.645,Z 620.222,A -85,B 0,C 180,E1 -25657.608,E2 -25657.608} C_VEL
LIN {X 0,Y 265.693,Z 620.987,A -85,B 0,C 180,E1 -25660.638,E2 -25660.638} C_VEL
LIN {X 0,Y 267.565,Z 620.453,A -85,B 0,C 180,E1 -25663.631,E2 -25663.631} C_VEL
LIN {X 0,Y 270.141,Z 618.634,A -85,B 0,C 180,E1 -25666.575,E2 -25666.575} C_VEL
LIN {X 0,Y 273.532,Z 615.501,A -85,B 0,C 180,E1 -25669.448,E2 -25669.448} C_VEL
LIN {X 0,Y 277.868,Z 610.973,A -85,B 0,C 180,E1 -25672.221,E2 -25672.221} C_VEL
LIN {X 0,Y 282.734,Z 604.999,A -85,B 0,C 180,E1 -25674.911,E2 -25674.911} C_VEL
LIN {X 0,Y 288.457,Z 597.3,A -85,B 0,C 180,E1 -25677.479,E2 -25677.479} C_VEL
LIN {X 0,Y 294.147,Z 588.955,A -85,B 0,C 180,E1 -25679.615,E2 -25679.615} C_VEL
LIN {X 0,Y 299.327,Z 580.495,A -85,B 0,C 180,E1 -25681.38,E2 -25681.38} C_VEL
LIN {X 0,Y 305.002,Z 570.399,A -85,B 0,C 180,E1 -25683.057,E2 -25683.057} C_VEL
LIN {X 0,Y 311.002,Z 558.374,A -85,B 0,C 180,E1 -25684.662,E2 -25684.662} C_VEL
LIN {X 0,Y 316.319,Z 546.299,A -85,B 0,C 180,E1 -25685.934,E2 -25685.934} C_VEL
LIN {X 0,Y 321.39,Z 532.991,A -85,B 0,C 180,E1 -25687.021,E2 -25687.021} C_VEL
LIN {X 0,Y 326.123,Z 518.281,A -85,B 0,C 180,E1 -25687.941,E2 -25687.941} C_VEL
LIN {X 0,Y 330.046,Z 502.867,A -85,B 0,C 180,E1 -25688.666,E2 -25688.666} C_VEL
LIN {X 0,Y 333.739,Z 482.065,A -85,B 0,C 180,E1 -25689.414,E2 -25689.414} C_VEL
LIN {X 0,Y 342.109,Z 431.364,A -85,B 0,C 180,E1 -25691.109,E2 -25691.109} C_VEL
LIN {X 0,Y 342.734,Z 424.195,A -85,B 0,C 180,E1 -25691.638,E2 -25691.638} C_VEL
LIN {X 0,Y 340.93,Z 420.478,A -85,B 0,C 180,E1 -25693.115,E2 -25693.115} C_VEL
LIN {X 0,Y 338.992,Z 416.76,A -85,B 0,C 180,E1 -25695.072,E2 -25695.072} C_VEL
LIN {X 0,Y 336.991,Z 413.355,A -85,B 0,C 180,E1 -25698.15,E2 -25698.15} C_VEL
LIN {X 0,Y 336.448,Z 412.575,A -85,B 0,C 180,E1 -25699.805,E2 -25699.805} C_VEL
LIN {X 0,Y 336.288,Z 412.965,A -85,B 0,C 180,E1 -25702.136,E2 -25702.136} C_VEL
LIN {X 0,Y 336.889,Z 414.941,A -85,B 0,C 180,E1 -25704.552,E2 -25704.552} C_VEL
LIN {X 0,Y 337.948,Z 417.649,A -85,B 0,C 180,E1 -25706.493,E2 -25706.493} C_VEL
LIN {X 0,Y 339.416,Z 421.513,A -85,B 0,C 180,E1 -25708.354,E2 -25708.354} C_VEL
LIN {X 0,Y 340.992,Z 426,A -85,B 0,C 180,E1 -25709.955,E2 -25709.955} C_VEL
LIN {X 0,Y 342.316,Z 430.099,A -85,B 0,C 180,E1 -25711.126,E2 -25711.126} C_VEL
LIN {X 0,Y 331.669,Z 493.712,A -85,B 0,C 180,E1 -25713.25,E2 -25713.25} C_VEL
LIN {X 0,Y 328.017,Z 509.341,A -85,B 0,C 180,E1 -25713.983,E2 -25713.983} C_VEL
LIN {X 0,Y 324.4,Z 521.739,A -85,B 0,C 180,E1 -25714.758,E2 -25714.758} C_VEL
LIN {X 0,Y 319.99,Z 534.518,A -85,B 0,C 180,E1 -25715.768,E2 -25715.768} C_VEL
LIN {X 0,Y 315.172,Z 546.419,A -85,B 0,C 180,E1 -25716.94,E2 -25716.94} C_VEL
LIN {X 0,Y 309.685,Z 558.194,A -85,B 0,C 180,E1 -25718.389,E2 -25718.389} C_VEL
LIN {X 0,Y 303.727,Z 569.354,A -85,B 0,C 180,E1 -25720.113,E2 -25720.113} C_VEL
LIN {X 0,Y 298.324,Z 578.461,A -85,B 0,C 180,E1 -25721.874,E2 -25721.874} C_VEL
LIN {X 0,Y 292.519,Z 587.259,A -85,B 0,C 180,E1 -25724.016,E2 -25724.016} C_VEL
LIN {X 0,Y 287.949,Z 593.48,A -85,B 0,C 180,E1 -25725.921,E2 -25725.921} C_VEL
LIN {X 0,Y 282.416,Z 600.235,A -85,B 0,C 180,E1 -25728.556,E2 -25728.556} C_VEL
LIN {X 0,Y 277.492,Z 605.346,A -85,B 0,C 180,E1 -25731.289,E2 -25731.289} C_VEL
LIN {X 0,Y 273.357,Z 608.937,A -85,B 0,C 180,E1 -25734.117,E2 -25734.117} C_VEL
LIN {X 0,Y 270.05,Z 611.139,A -85,B 0,C 180,E1 -25737.026,E2 -25737.026} C_VEL
LIN {X 0,Y 267.585,Z 612.001,A -85,B 0,C 180,E1 -25740,E2 -25740} C_VEL
LIN {X 0,Y 265.843,Z 611.495,A -85,B 0,C 180,E1 -25743.124,E2 -25743.124} C_VEL
LIN {X 0,Y 264.724,Z 609.747,A -85,B 0,C 180,E1 -25746.075,E2 -25746.075} C_VEL
LIN {X 0,Y 264.213,Z 606.561,A -85,B 0,C 180,E1 -25749.152,E2 -25749.152} C_VEL
LIN {X 0,Y 264.153,Z 603.721,A -85,B 0,C 180,E1 -25751.138,E2 -25751.138} C_VEL
LIN {X 0,Y 264.164,Z 598.812,A -85,B 0,C 180,E1 -25753.806,E2 -25753.806} C_VEL
LIN {X 0,Y 264.474,Z 592.34,A -85,B 0,C 180,E1 -25756.541,E2 -25756.541} C_VEL
LIN {X 0,Y 264.9,Z 584.094,A -85,B 0,C 180,E1 -25759.3,E2 -25759.3} C_VEL
LIN {X 0,Y 265.445,Z 575.357,A -85,B 0,C 180,E1 -25761.68,E2 -25761.68} C_VEL
LIN {X 0,Y 266.21,Z 564.712,A -85,B 0,C 180,E1 -25764.069,E2 -25764.069} C_VEL
LIN {X 0,Y 267.101,Z 553.902,A -85,B 0,C 180,E1 -25766.056,E2 -25766.056} C_VEL
LIN {X 0,Y 268.219,Z 540.772,A -85,B 0,C 180,E1 -25768.038,E2 -25768.038} C_VEL
LIN {X 0,Y 269.235,Z 527.865,A -85,B 0,C 180,E1 -25769.624,E2 -25769.624} C_VEL
LIN {X 0,Y 270.32,Z 513.814,A -85,B 0,C 180,E1 -25770.997,E2 -25770.997} C_VEL
LIN {X 0,Y 271.335,Z 498.878,A -85,B 0,C 180,E1 -25772.114,E2 -25772.114} C_VEL
LIN {X 0,Y 272.224,Z 483.933,A -85,B 0,C 180,E1 -25772.926,E2 -25772.926} C_VEL
LIN {X 0,Y 276.078,Z 388.32,A -85,B 0,C 180,E1 -25776.713,E2 -25776.713} C_VEL
LIN {X 0,Y 273.239,Z 359.593,A -85,B 0,C 180,E1 -25777.986,E2 -25777.986} C_VEL
LIN {X 0,Y 272.443,Z 348.92,A -85,B 0,C 180,E1 -25778.457,E2 -25778.457} C_VEL
LIN {X 0,Y 271.945,Z 346.649,A -85,B 0,C 180,E1 -25778.613,E2 -25778.613} C_VEL
LIN {X 0,Y 268.226,Z 328.104,A -85,B 0,C 180,E1 -25782.763,E2 -25782.763} C_VEL
LIN {X 0,Y 267.311,Z 323.747,A -85,B 0,C 180,E1 -25783.757,E2 -25783.757} C_VEL
LIN {X 0,Y 267.266,Z 323.749,A -85,B 0,C 180,E1 -25787.207,E2 -25787.207} C_VEL
LIN {X 0,Y 267.235,Z 323.752,A -85,B 0,C 180,E1 -25791.015,E2 -25791.015} C_VEL
LIN {X 0,Y 267.296,Z 323.734,A -85,B 0,C 180,E1 -25794.791,E2 -25794.791} C_VEL
LIN {X 0,Y 267.268,Z 323.749,A -85,B 0,C 180,E1 -25798.385,E2 -25798.385} C_VEL
LIN {X 0,Y 267.301,Z 323.734,A -85,B 0,C 180,E1 -25801.853,E2 -25801.853} C_VEL
LIN {X 0,Y 267.289,Z 323.748,A -85,B 0,C 180,E1 -25805.207,E2 -25805.207} C_VEL
LIN {X 0,Y 267.349,Z 323.742,A -85,B 0,C 180,E1 -25808.478,E2 -25808.478} C_VEL
LIN {X 0,Y 267.407,Z 323.735,A -85,B 0,C 180,E1 -25810.195,E2 -25810.195} C_VEL
LIN {X 0,Y 268.506,Z 326.713,A -85,B 0,C 180,E1 -25810.409,E2 -25810.409} C_VEL
LIN {X 0,Y 275.722,Z 341.527,A -85,B 0,C 180,E1 -25811.598,E2 -25811.598} C_VEL
LIN {X 0,Y 282.837,Z 358.31,A -85,B 0,C 180,E1 -25812.765,E2 -25812.765} C_VEL
LIN {X 0,Y 284.136,Z 362.319,A -85,B 0,C 180,E1 -25812.997,E2 -25812.997} C_VEL
LIN {X 0,Y 281.17,Z 452.636,A -85,B 0,C 180,E1 -25815.249,E2 -25815.249} C_VEL
LIN {X 0,Y 280.285,Z 466.369,A -85,B 0,C 180,E1 -25815.848,E2 -25815.848} C_VEL
LIN {X 0,Y 279.131,Z 480.386,A -85,B 0,C 180,E1 -25816.76,E2 -25816.76} C_VEL
LIN {X 0,Y 277.798,Z 492.53,A -85,B 0,C 180,E1 -25817.806,E2 -25817.806} C_VEL
LIN {X 0,Y 276.165,Z 503.927,A -85,B 0,C 180,E1 -25819.031,E2 -25819.031} C_VEL
LIN {X 0,Y 274.165,Z 515.84,A -85,B 0,C 180,E1 -25820.623,E2 -25820.623} C_VEL
LIN {X 0,Y 272.634,Z 525.685,A -85,B 0,C 180,E1 -25822.245,E2 -25822.245} C_VEL
LIN {X 0,Y 270.947,Z 534.937,A -85,B 0,C 180,E1 -25824.061,E2 -25824.061} C_VEL
LIN {X 0,Y 269.171,Z 544.219,A -85,B 0,C 180,E1 -25826.266,E2 -25826.266} C_VEL
LIN {X 0,Y 267.668,Z 551.951,A -85,B 0,C 180,E1 -25828.497,E2 -25828.497} C_VEL
LIN {X 0,Y 266.751,Z 558.336,A -85,B 0,C 180,E1 -25830.749,E2 -25830.749} C_VEL
LIN {X 0,Y 266,Z 563.646,A -85,B 0,C 180,E1 -25833.015,E2 -25833.015} C_VEL
LIN {X 0,Y 265.312,Z 568.028,A -85,B 0,C 180,E1 -25835.298,E2 -25835.298} C_VEL
LIN {X 0,Y 264.797,Z 571.518,A -85,B 0,C 180,E1 -25837.596,E2 -25837.596} C_VEL
LIN {X 0,Y 264.631,Z 574.864,A -85,B 0,C 180,E1 -25840.674,E2 -25840.674} C_VEL
LIN {X 0,Y 264.732,Z 576.811,A -85,B 0,C 180,E1 -25843.772,E2 -25843.772} C_VEL
LIN {X 0,Y 265.299,Z 577.399,A -85,B 0,C 180,E1 -25846.879,E2 -25846.879} C_VEL
LIN {X 0,Y 266.336,Z 576.628,A -85,B 0,C 180,E1 -25849.988,E2 -25849.988} C_VEL
LIN {X 0,Y 267.935,Z 574.467,A -85,B 0,C 180,E1 -25853.083,E2 -25853.083} C_VEL
LIN {X 0,Y 270.157,Z 570.842,A -85,B 0,C 180,E1 -25856.148,E2 -25856.148} C_VEL
LIN {X 0,Y 272.967,Z 565.634,A -85,B 0,C 180,E1 -25859.175,E2 -25859.175} C_VEL
LIN {X 0,Y 275.556,Z 560.517,A -85,B 0,C 180,E1 -25861.401,E2 -25861.401} C_VEL
LIN {X 0,Y 278.48,Z 554.28,A -85,B 0,C 180,E1 -25863.592,E2 -25863.592} C_VEL
LIN {X 0,Y 281.734,Z 546.727,A -85,B 0,C 180,E1 -25865.745,E2 -25865.745} C_VEL
LIN {X 0,Y 285.338,Z 537.582,A -85,B 0,C 180,E1 -25867.852,E2 -25867.852} C_VEL
LIN {X 0,Y 288.648,Z 528.422,A -85,B 0,C 180,E1 -25869.563,E2 -25869.563} C_VEL
LIN {X 0,Y 292.141,Z 517.407,A -85,B 0,C 180,E1 -25871.245,E2 -25871.245} C_VEL
LIN {X 0,Y 295.168,Z 506.164,A -85,B 0,C 180,E1 -25872.639,E2 -25872.639} C_VEL
LIN {X 0,Y 298.021,Z 493.518,A -85,B 0,C 180,E1 -25873.89,E2 -25873.89} C_VEL
LIN {X 0,Y 300.465,Z 479.601,A -85,B 0,C 180,E1 -25874.957,E2 -25874.957} C_VEL
LIN {X 0,Y 302.319,Z 465.634,A -85,B 0,C 180,E1 -25875.725,E2 -25875.725} C_VEL
LIN {X 0,Y 303.482,Z 452.505,A -85,B 0,C 180,E1 -25876.221,E2 -25876.221} C_VEL
LIN {X 0,Y 306.687,Z 387.614,A -85,B 0,C 180,E1 -25877.72,E2 -25877.72} C_VEL
LIN {X 0,Y 298.818,Z 371.364,A -85,B 0,C 180,E1 -25879.57,E2 -25879.57} C_VEL
LIN {X 0,Y 290.549,Z 357.555,A -85,B 0,C 180,E1 -25881.584,E2 -25881.584} C_VEL
LIN {X 0,Y 282.243,Z 345.181,A -85,B 0,C 180,E1 -25883.754,E2 -25883.754} C_VEL
LIN {X 0,Y 276.947,Z 337.712,A -85,B 0,C 180,E1 -25885.242,E2 -25885.242} C_VEL
LIN {X 0,Y 273.885,Z 333.511,A -85,B 0,C 180,E1 -25886.149,E2 -25886.149} C_VEL
LIN {X 0,Y 271.46,Z 330.446,A -85,B 0,C 180,E1 -25886.883,E2 -25886.883} C_VEL
LIN {X 0,Y 270.528,Z 328.871,A -85,B 0,C 180,E1 -25887.188,E2 -25887.188} C_VEL
LIN {X 0,Y 268.33,Z 326.705,A -85,B 0,C 180,E1 -25887.86,E2 -25887.86} C_VEL
LIN {X 0,Y 267.326,Z 324.205,A -85,B 0,C 180,E1 -25888.239,E2 -25888.239} C_VEL
LIN {X 0,Y 267.249,Z 323.745,A -85,B 0,C 180,E1 -25888.308,E2 -25888.308} C_VEL
LIN {X 0,Y 267.288,Z 323.738,A -85,B 0,C 180,E1 -25891.855,E2 -25891.855} C_VEL
LIN {X 0,Y 267.29,Z 323.744,A -85,B 0,C 180,E1 -25895.21,E2 -25895.21} C_VEL
LIN {X 0,Y 267.307,Z 323.745,A -85,B 0,C 180,E1 -25898.478,E2 -25898.478} C_VEL
LIN {X 0,Y 267.377,Z 323.721,A -85,B 0,C 180,E1 -25901.678,E2 -25901.678} C_VEL
LIN {X 0,Y 267.524,Z 323.699,A -85,B 0,C 180,E1 -25906.371,E2 -25906.371} C_VEL
LIN {X 0,Y 267.61,Z 323.686,A -85,B 0,C 180,E1 -25910.965,E2 -25910.965} C_VEL
LIN {X 0,Y 267.794,Z 323.685,A -85,B 0,C 180,E1 -25913.995,E2 -25913.995} C_VEL
LIN {X 0,Y 267.89,Z 323.671,A -85,B 0,C 180,E1 -25918.502,E2 -25918.502} C_VEL
LIN {X 0,Y 267.89,Z 323.649,A -85,B 0,C 180,E1 -25921.498,E2 -25921.498} C_VEL
LIN {X 0,Y 267.794,Z 323.67,A -85,B 0,C 180,E1 -25926.006,E2 -25926.006} C_VEL
LIN {X 0,Y 267.559,Z 323.708,A -85,B 0,C 180,E1 -25930.559,E2 -25930.559} C_VEL
LIN {X 0,Y 267.534,Z 323.708,A -85,B 0,C 180,E1 -25934.388,E2 -25934.388} C_VEL
LIN {X 0,Y 267.409,Z 323.727,A -85,B 0,C 180,E1 -25939.456,E2 -25939.456} C_VEL
LIN {X 0,Y 267.387,Z 323.733,A -85,B 0,C 180,E1 -25939.828,E2 -25939.828} C_VEL
LIN {X 0,Y 266.676,Z 323.828,A -85,B 0,C 180,E1 -25941.084,E2 -25941.084} C_VEL
LIN {X 0,Y 263.766,Z 324.186,A -85,B 0,C 180,E1 -25943.131,E2 -25943.131} C_VEL
LIN {X 0,Y 261.329,Z 324.489,A -85,B 0,C 180,E1 -25944.795,E2 -25944.795} C_VEL
LIN {X 0,Y 260.305,Z 324.604,A -85,B 0,C 180,E1 -25946.087,E2 -25946.087} C_VEL
LIN {X 0,Y 260.232,Z 324.612,A -85,B 0,C 180,E1 -25946.524,E2 -25946.524} C_VEL
LIN {X 0,Y 260.212,Z 324.617,A -85,B 0,C 180,E1 -25950.76,E2 -25950.76} C_VEL
LIN {X 0,Y 260.231,Z 324.587,A -85,B 0,C 180,E1 -25954.419,E2 -25954.419} C_VEL
LIN {X 0,Y 262.129,Z 330.263,A -85,B 0,C 180,E1 -25957.922,E2 -25957.922} C_VEL
LIN {X 0,Y 264.173,Z 336.837,A -85,B 0,C 180,E1 -25961.519,E2 -25961.519} C_VEL
LIN {X 0,Y 265.219,Z 340.102,A -85,B 0,C 180,E1 -25963.12,E2 -25963.12} C_VEL
LIN {X 0,Y 268.068,Z 344.859,A -85,B 0,C 180,E1 -25964.086,E2 -25964.086} C_VEL
LIN {X 0,Y 269.762,Z 347.44,A -85,B 0,C 180,E1 -25964.632,E2 -25964.632} C_VEL
LIN {X 0,Y 273.26,Z 353.136,A -85,B 0,C 180,E1 -25965.732,E2 -25965.732} C_VEL
LIN {X 0,Y 276.948,Z 359.435,A -85,B 0,C 180,E1 -25966.845,E2 -25966.845} C_VEL
LIN {X 0,Y 282.288,Z 368.867,A -85,B 0,C 180,E1 -25968.374,E2 -25968.374} C_VEL
LIN {X 0,Y 289.624,Z 383.437,A -85,B 0,C 180,E1 -25970.375,E2 -25970.375} C_VEL
LIN {X 0,Y 296.201,Z 398.575,A -85,B 0,C 180,E1 -25972.096,E2 -25972.096} C_VEL
LIN {X 0,Y 298.707,Z 417.139,A -85,B 0,C 180,E1 -25973.126,E2 -25973.126} C_VEL
LIN {X 0,Y 299.612,Z 425.362,A -85,B 0,C 180,E1 -25973.537,E2 -25973.537} C_VEL
LIN {X 0,Y 296.561,Z 481.262,A -85,B 0,C 180,E1 -25974.834,E2 -25974.834} C_VEL
LIN {X 0,Y 294.906,Z 495.937,A -85,B 0,C 180,E1 -25975.407,E2 -25975.407} C_VEL
LIN {X 0,Y 292.467,Z 509.733,A -85,B 0,C 180,E1 -25976.168,E2 -25976.168} C_VEL
LIN {X 0,Y 289.276,Z 523.508,A -85,B 0,C 180,E1 -25977.2,E2 -25977.2} C_VEL
LIN {X 0,Y 285.914,Z 535.859,A -85,B 0,C 180,E1 -25978.427,E2 -25978.427} C_VEL
LIN {X 0,Y 281.902,Z 548.347,A -85,B 0,C 180,E1 -25980.001,E2 -25980.001} C_VEL
LIN {X 0,Y 278.016,Z 559.424,A -85,B 0,C 180,E1 -25981.793,E2 -25981.793} C_VEL
LIN {X 0,Y 273.97,Z 569.561,A -85,B 0,C 180,E1 -25983.835,E2 -25983.835} C_VEL
LIN {X 0,Y 270.352,Z 577.939,A -85,B 0,C 180,E1 -25985.921,E2 -25985.921} C_VEL
LIN {X 0,Y 266.648,Z 585.982,A -85,B 0,C 180,E1 -25988.427,E2 -25988.427} C_VEL
LIN {X 0,Y 264.071,Z 591.685,A -85,B 0,C 180,E1 -25990.641,E2 -25990.641} C_VEL
LIN {X 0,Y 261.331,Z 597.718,A -85,B 0,C 180,E1 -25993.659,E2 -25993.659} C_VEL
LIN {X 0,Y 259.447,Z 601.806,A -85,B 0,C 180,E1 -25996.389,E2 -25996.389} C_VEL
LIN {X 0,Y 258.195,Z 604.672,A -85,B 0,C 180,E1 -25999.057,E2 -25999.057} C_VEL
LIN {X 0,Y 257.392,Z 606.754,A -85,B 0,C 180,E1 -26002.184,E2 -26002.184} C_VEL
LIN {X 0,Y 257.427,Z 607.538,A -85,B 0,C 180,E1 -26005.322,E2 -26005.322} C_VEL
LIN {X 0,Y 257.894,Z 607.216,A -85,B 0,C 180,E1 -26007.864,E2 -26007.864} C_VEL
LIN {X 0,Y 257.77,Z 611.322,A -85,B 0,C 180,E1 -26010.004,E2 -26010.004} C_VEL
LIN {X 0,Y 257.533,Z 614.816,A -85,B 0,C 180,E1 -26012.342,E2 -26012.342} C_VEL
LIN {X 0,Y 257.394,Z 617.476,A -85,B 0,C 180,E1 -26014.686,E2 -26014.686} C_VEL
LIN {X 0,Y 257.605,Z 619.769,A -85,B 0,C 180,E1 -26017.817,E2 -26017.817} C_VEL
LIN {X 0,Y 258.697,Z 620.765,A -85,B 0,C 180,E1 -26020.929,E2 -26020.929} C_VEL
LIN {X 0,Y 260.665,Z 620.48,A -85,B 0,C 180,E1 -26023.999,E2 -26023.999} C_VEL
LIN {X 0,Y 263.352,Z 618.915,A -85,B 0,C 180,E1 -26027.015,E2 -26027.015} C_VEL
LIN {X 0,Y 266.87,Z 616.061,A -85,B 0,C 180,E1 -26029.954,E2 -26029.954} C_VEL
LIN {X 0,Y 271.38,Z 611.833,A -85,B 0,C 180,E1 -26032.781,E2 -26032.781} C_VEL
LIN {X 0,Y 276.404,Z 606.183,A -85,B 0,C 180,E1 -26035.522,E2 -26035.522} C_VEL
LIN {X 0,Y 282.32,Z 598.919,A -85,B 0,C 180,E1 -26038.128,E2 -26038.128} C_VEL
LIN {X 0,Y 288.181,Z 591.046,A -85,B 0,C 180,E1 -26040.291,E2 -26040.291} C_VEL
LIN {X 0,Y 294.451,Z 581.534,A -85,B 0,C 180,E1 -26042.363,E2 -26042.363} C_VEL
LIN {X 0,Y 300.355,Z 571.682,A -85,B 0,C 180,E1 -26044.038,E2 -26044.038} C_VEL
LIN {X 0,Y 306.054,Z 561.054,A -85,B 0,C 180,E1 -26045.506,E2 -26045.506} C_VEL
LIN {X 0,Y 312.036,Z 548.321,A -85,B 0,C 180,E1 -26046.907,E2 -26046.907} C_VEL
LIN {X 0,Y 317.263,Z 535.665,A -85,B 0,C 180,E1 -26047.985,E2 -26047.985} C_VEL
LIN {X 0,Y 322.075,Z 521.785,A -85,B 0,C 180,E1 -26048.904,E2 -26048.904} C_VEL
LIN {X 0,Y 326.44,Z 506.31,A -85,B 0,C 180,E1 -26049.672,E2 -26049.672} C_VEL
LIN {X 0,Y 329.771,Z 490.249,A -85,B 0,C 180,E1 -26050.282,E2 -26050.282} C_VEL
LIN {X 0,Y 339.58,Z 433.036,A -85,B 0,C 180,E1 -26052.193,E2 -26052.193} C_VEL
LIN {X 0,Y 339.94,Z 429.185,A -85,B 0,C 180,E1 -26052.501,E2 -26052.501} C_VEL
LIN {X 0,Y 337.688,Z 424.498,A -85,B 0,C 180,E1 -26054.677,E2 -26054.677} C_VEL
LIN {X 0,Y 336.449,Z 422.338,A -85,B 0,C 180,E1 -26056.208,E2 -26056.208} C_VEL
LIN {X 0,Y 335.157,Z 419.848,A -85,B 0,C 180,E1 -26058.799,E2 -26058.799} C_VEL
LIN {X 0,Y 334.721,Z 419.492,A -85,B 0,C 180,E1 -26060.742,E2 -26060.742} C_VEL
LIN {X 0,Y 334.785,Z 420.334,A -85,B 0,C 180,E1 -26062.821,E2 -26062.821} C_VEL
LIN {X 0,Y 335.465,Z 422.573,A -85,B 0,C 180,E1 -26065.025,E2 -26065.025} C_VEL
LIN {X 0,Y 336.259,Z 424.697,A -85,B 0,C 180,E1 -26066.435,E2 -26066.435} C_VEL
LIN {X 0,Y 337.45,Z 428.151,A -85,B 0,C 180,E1 -26068.056,E2 -26068.056} C_VEL
LIN {X 0,Y 339.103,Z 433.251,A -85,B 0,C 180,E1 -26069.845,E2 -26069.845} C_VEL
LIN {X 0,Y 339.348,Z 434.175,A -85,B 0,C 180,E1 -26070.106,E2 -26070.106} C_VEL
LIN {X 0,Y 328.981,Z 493.836,A -85,B 0,C 180,E1 -26072.112,E2 -26072.112} C_VEL
LIN {X 0,Y 325.403,Z 508.585,A -85,B 0,C 180,E1 -26072.779,E2 -26072.779} C_VEL
LIN {X 0,Y 321.195,Z 522.445,A -85,B 0,C 180,E1 -26073.632,E2 -26073.632} C_VEL
LIN {X 0,Y 316.219,Z 536.158,A -85,B 0,C 180,E1 -26074.726,E2 -26074.726} C_VEL
LIN {X 0,Y 310.557,Z 549.119,A -85,B 0,C 180,E1 -26076.047,E2 -26076.047} C_VEL
LIN {X 0,Y 304.803,Z 560.617,A -85,B 0,C 180,E1 -26077.515,E2 -26077.515} C_VEL
LIN {X 0,Y 298.252,Z 572.1,A -85,B 0,C 180,E1 -26079.373,E2 -26079.373} C_VEL
LIN {X 0,Y 292.677,Z 580.763,A -85,B 0,C 180,E1 -26081.15,E2 -26081.15} C_VEL
LIN {X 0,Y 286.661,Z 589.14,A -85,B 0,C 180,E1 -26083.315,E2 -26083.315} C_VEL
LIN {X 0,Y 281.137,Z 595.978,A -85,B 0,C 180,E1 -26085.573,E2 -26085.573} C_VEL
LIN {X 0,Y 275.48,Z 602.151,A -85,B 0,C 180,E1 -26088.263,E2 -26088.263} C_VEL
LIN {X 0,Y 270.455,Z 606.795,A -85,B 0,C 180,E1 -26091.06,E2 -26091.06} C_VEL
LIN {X 0,Y 266.285,Z 609.961,A -85,B 0,C 180,E1 -26093.96,E2 -26093.96} C_VEL
LIN {X 0,Y 262.897,Z 611.759,A -85,B 0,C 180,E1 -26096.945,E2 -26096.945} C_VEL
LIN {X 0,Y 260.429,Z 612.227,A -85,B 0,C 180,E1 -26100,E2 -26100} C_VEL
LIN {X 0,Y 258.723,Z 611.379,A -85,B 0,C 180,E1 -26103.104,E2 -26103.104} C_VEL
LIN {X 0,Y 257.584,Z 609.184,A -85,B 0,C 180,E1 -26106.244,E2 -26106.244} C_VEL
LIN {X 0,Y 257.133,Z 605.577,A -85,B 0,C 180,E1 -26109.407,E2 -26109.407} C_VEL
LIN {X 0,Y 257.054,Z 601.892,A -85,B 0,C 180,E1 -26111.792,E2 -26111.792} C_VEL
LIN {X 0,Y 257.162,Z 597.153,A -85,B 0,C 180,E1 -26114.19,E2 -26114.19} C_VEL
LIN {X 0,Y 257.472,Z 590.233,A -85,B 0,C 180,E1 -26117.005,E2 -26117.005} C_VEL
LIN {X 0,Y 257.862,Z 582.836,A -85,B 0,C 180,E1 -26119.436,E2 -26119.436} C_VEL
LIN {X 0,Y 258.455,Z 573.799,A -85,B 0,C 180,E1 -26121.879,E2 -26121.879} C_VEL
LIN {X 0,Y 259.261,Z 562.712,A -85,B 0,C 180,E1 -26124.331,E2 -26124.331} C_VEL
LIN {X 0,Y 260.294,Z 550.33,A -85,B 0,C 180,E1 -26126.575,E2 -26126.575} C_VEL
LIN {X 0,Y 261.346,Z 537.745,A -85,B 0,C 180,E1 -26128.429,E2 -26128.429} C_VEL
LIN {X 0,Y 262.443,Z 524.304,A -85,B 0,C 180,E1 -26130.028,E2 -26130.028} C_VEL
LIN {X 0,Y 263.515,Z 509.696,A -85,B 0,C 180,E1 -26131.402,E2 -26131.402} C_VEL
LIN {X 0,Y 264.496,Z 495.189,A -85,B 0,C 180,E1 -26132.43,E2 -26132.43} C_VEL
LIN {X 0,Y 265.304,Z 479.5,A -85,B 0,C 180,E1 -26133.218,E2 -26133.218} C_VEL
LIN {X 0,Y 269.124,Z 389.402,A -85,B 0,C 180,E1 -26136.905,E2 -26136.905} C_VEL
LIN {X 0,Y 266.31,Z 360.781,A -85,B 0,C 180,E1 -26138.204,E2 -26138.204} C_VEL
LIN {X 0,Y 265.387,Z 349.592,A -85,B 0,C 180,E1 -26138.713,E2 -26138.713} C_VEL
LIN {X 0,Y 264.785,Z 347.002,A -85,B 0,C 180,E1 -26138.853,E2 -26138.853} C_VEL
LIN {X 0,Y 261.098,Z 328.65,A -85,B 0,C 180,E1 -26143.039,E2 -26143.039} C_VEL
LIN {X 0,Y 260.261,Z 324.623,A -85,B 0,C 180,E1 -26144,E2 -26144} C_VEL
LIN {X 0,Y 260.231,Z 324.624,A -85,B 0,C 180,E1 -26148.908,E2 -26148.908} C_VEL
LIN {X 0,Y 260.192,Z 324.63,A -85,B 0,C 180,E1 -26151.741,E2 -26151.741} C_VEL
LIN {X 0,Y 260.229,Z 324.609,A -85,B 0,C 180,E1 -26155.577,E2 -26155.577} C_VEL
LIN {X 0,Y 260.206,Z 324.63,A -85,B 0,C 180,E1 -26159.475,E2 -26159.475} C_VEL
LIN {X 0,Y 260.275,Z 324.611,A -85,B 0,C 180,E1 -26162.77,E2 -26162.77} C_VEL
LIN {X 0,Y 260.304,Z 324.618,A -85,B 0,C 180,E1 -26166.191,E2 -26166.191} C_VEL
LIN {X 0,Y 260.333,Z 324.646,A -85,B 0,C 180,E1 -26169.42,E2 -26169.42} C_VEL
LIN {X 0,Y 261.296,Z 327.413,A -85,B 0,C 180,E1 -26169.618,E2 -26169.618} C_VEL
LIN {X 0,Y 267.591,Z 339.812,A -85,B 0,C 180,E1 -26170.698,E2 -26170.698} C_VEL
LIN {X 0,Y 275.743,Z 358.293,A -85,B 0,C 180,E1 -26172.079,E2 -26172.079} C_VEL
LIN {X 0,Y 277.63,Z 363.727,A -85,B 0,C 180,E1 -26172.418,E2 -26172.418} C_VEL
LIN {X 0,Y 274.613,Z 453.152,A -85,B 0,C 180,E1 -26174.699,E2 -26174.699} C_VEL
LIN {X 0,Y 273.705,Z 466.845,A -85,B 0,C 180,E1 -26175.311,E2 -26175.311} C_VEL
LIN {X 0,Y 272.514,Z 480.843,A -85,B 0,C 180,E1 -26176.243,E2 -26176.243} C_VEL
LIN {X 0,Y 271.141,Z 492.975,A -85,B 0,C 180,E1 -26177.312,E2 -26177.312} C_VEL
LIN {X 0,Y 269.448,Z 504.368,A -85,B 0,C 180,E1 -26178.564,E2 -26178.564} C_VEL
LIN {X 0,Y 267.391,Z 516.274,A -85,B 0,C 180,E1 -26180.193,E2 -26180.193} C_VEL
LIN {X 0,Y 265.621,Z 527.087,A -85,B 0,C 180,E1 -26182.039,E2 -26182.039} C_VEL
LIN {X 0,Y 263.88,Z 536.189,A -85,B 0,C 180,E1 -26183.901,E2 -26183.901} C_VEL
LIN {X 0,Y 262.117,Z 545.316,A -85,B 0,C 180,E1 -26186.166,E2 -26186.166} C_VEL
LIN {X 0,Y 260.545,Z 552.945,A -85,B 0,C 180,E1 -26188.456,E2 -26188.456} C_VEL
LIN {X 0,Y 259.65,Z 559.26,A -85,B 0,C 180,E1 -26190.769,E2 -26190.769} C_VEL
LIN {X 0,Y 258.884,Z 564.472,A -85,B 0,C 180,E1 -26193.098,E2 -26193.098} C_VEL
LIN {X 0,Y 258.178,Z 568.762,A -85,B 0,C 180,E1 -26195.445,E2 -26195.445} C_VEL
LIN {X 0,Y 257.675,Z 572.2,A -85,B 0,C 180,E1 -26197.808,E2 -26197.808} C_VEL
LIN {X 0,Y 257.547,Z 575.431,A -85,B 0,C 180,E1 -26200.971,E2 -26200.971} C_VEL
LIN {X 0,Y 257.678,Z 577.295,A -85,B 0,C 180,E1 -26204.157,E2 -26204.157} C_VEL
LIN {X 0,Y 258.322,Z 577.802,A -85,B 0,C 180,E1 -26207.349,E2 -26207.349} C_VEL
LIN {X 0,Y 259.466,Z 576.948,A -85,B 0,C 180,E1 -26210.541,E2 -26210.541} C_VEL
LIN {X 0,Y 261.206,Z 574.701,A -85,B 0,C 180,E1 -26213.714,E2 -26213.714} C_VEL
LIN {X 0,Y 263.594,Z 570.988,A -85,B 0,C 180,E1 -26216.851,E2 -26216.851} C_VEL
LIN {X 0,Y 266.458,Z 565.887,A -85,B 0,C 180,E1 -26219.833,E2 -26219.833} C_VEL
LIN {X 0,Y 269.804,Z 559.493,A -85,B 0,C 180,E1 -26222.59,E2 -26222.59} C_VEL
LIN {X 0,Y 273.556,Z 551.579,A -85,B 0,C 180,E1 -26225.225,E2 -26225.225} C_VEL
LIN {X 0,Y 277.024,Z 543.548,A -85,B 0,C 180,E1 -26227.356,E2 -26227.356} C_VEL
LIN {X 0,Y 280.589,Z 534.529,A -85,B 0,C 180,E1 -26229.298,E2 -26229.298} C_VEL
LIN {X 0,Y 284.435,Z 523.594,A -85,B 0,C 180,E1 -26231.198,E2 -26231.198} C_VEL
LIN {X 0,Y 288.151,Z 511.403,A -85,B 0,C 180,E1 -26232.887,E2 -26232.887} C_VEL
LIN {X 0,Y 291.255,Z 499.31,A -85,B 0,C 180,E1 -26234.215,E2 -26234.215} C_VEL
LIN {X 0,Y 293.939,Z 485.859,A -85,B 0,C 180,E1 -26235.385,E2 -26235.385} C_VEL
LIN {X 0,Y 296.038,Z 472.514,A -85,B 0,C 180,E1 -26236.246,E2 -26236.246} C_VEL
LIN {X 0,Y 297.585,Z 458.337,A -85,B 0,C 180,E1 -26236.896,E2 -26236.896} C_VEL
LIN {X 0,Y 298.683,Z 440.38,A -85,B 0,C 180,E1 -26237.395,E2 -26237.395} C_VEL
LIN {X 0,Y 301.328,Z 390.192,A -85,B 0,C 180,E1 -26238.531,E2 -26238.531} C_VEL
LIN {X 0,Y 294.109,Z 375.212,A -85,B 0,C 180,E1 -26240.301,E2 -26240.301} C_VEL
LIN {X 0,Y 286.017,Z 361.728,A -85,B 0,C 180,E1 -26242.352,E2 -26242.352} C_VEL
LIN {X 0,Y 278.568,Z 350.442,A -85,B 0,C 180,E1 -26244.377,E2 -26244.377} C_VEL
LIN {X 0,Y 273.425,Z 343.113,A -85,B 0,C 180,E1 -26245.878,E2 -26245.878} C_VEL
LIN {X 0,Y 270.196,Z 338.774,A -85,B 0,C 180,E1 -26246.864,E2 -26246.864} C_VEL
LIN {X 0,Y 267.64,Z 335.089,A -85,B 0,C 180,E1 -26247.688,E2 -26247.688} C_VEL
LIN {X 0,Y 264.897,Z 331.938,A -85,B 0,C 180,E1 -26248.573,E2 -26248.573} C_VEL
LIN {X 0,Y 263.805,Z 329.948,A -85,B 0,C 180,E1 -26248.969,E2 -26248.969} C_VEL
LIN {X 0,Y 261.596,Z 328.026,A -85,B 0,C 180,E1 -26249.694,E2 -26249.694} C_VEL
LIN {X 0,Y 260.419,Z 325.509,A -85,B 0,C 180,E1 -26250.159,E2 -26250.159} C_VEL
LIN {X 0,Y 260.247,Z 324.621,A -85,B 0,C 180,E1 -26250.304,E2 -26250.304} C_VEL
LIN {X 0,Y 260.25,Z 324.626,A -85,B 0,C 180,E1 -26254.493,E2 -26254.493} C_VEL
LIN {X 0,Y 260.284,Z 324.61,A -85,B 0,C 180,E1 -26257.868,E2 -26257.868} C_VEL
LIN {X 0,Y 260.334,Z 324.596,A -85,B 0,C 180,E1 -26261.164,E2 -26261.164} C_VEL
LIN {X 0,Y 260.46,Z 324.578,A -85,B 0,C 180,E1 -26265.993,E2 -26265.993} C_VEL
LIN {X 0,Y 260.54,Z 324.567,A -85,B 0,C 180,E1 -26270.717,E2 -26270.717} C_VEL
LIN {X 0,Y 260.761,Z 324.562,A -85,B 0,C 180,E1 -26273.832,E2 -26273.832} C_VEL
LIN {X 0,Y 260.842,Z 324.548,A -85,B 0,C 180,E1 -26278.461,E2 -26278.461} C_VEL
LIN {X 0,Y 260.957,Z 324.53,A -85,B 0,C 180,E1 -26280,E2 -26280} C_VEL
LIN {X 0,Y 260.782,Z 324.559,A -85,B 0,C 180,E1 -26284.622,E2 -26284.622} C_VEL
LIN {X 0,Y 260.626,Z 324.553,A -85,B 0,C 180,E1 -26287.723,E2 -26287.723} C_VEL
LIN {X 0,Y 260.461,Z 324.573,A -85,B 0,C 180,E1 -26292.424,E2 -26292.424} C_VEL
LIN {X 0,Y 260.372,Z 324.604,A -85,B 0,C 180,E1 -26295.606,E2 -26295.606} C_VEL
LIN {X 0,Y 260.347,Z 324.609,A -85,B 0,C 180,E1 -26299.793,E2 -26299.793} C_VEL
LIN {X 0,Y 260.279,Z 324.615,A -85,B 0,C 180,E1 -26303.808,E2 -26303.808} C_VEL
LIN {X 0,Y 260.232,Z 324.612,A -85,B 0,C 180,E1 -26306.524,E2 -26306.524} C_VEL
LIN {X 0,Y 259.572,Z 324.699,A -85,B 0,C 180,E1 -26307.385,E2 -26307.385} C_VEL
LIN {X 0,Y 256.741,Z 325.063,A -85,B 0,C 180,E1 -26308.735,E2 -26308.735} C_VEL
LIN {X 0,Y 253.862,Z 325.411,A -85,B 0,C 180,E1 -26310.113,E2 -26310.113} C_VEL
LIN {X 0,Y 253.167,Z 325.495,A -85,B 0,C 180,E1 -26311.006,E2 -26311.006} C_VEL
LIN {X 0,Y 253.216,Z 325.641,A -85,B 0,C 180,E1 -26312.526,E2 -26312.526} C_VEL
LIN {X 0,Y 255.109,Z 331.079,A -85,B 0,C 180,E1 -26316.18,E2 -26316.18} C_VEL
LIN {X 0,Y 257.332,Z 338.198,A -85,B 0,C 180,E1 -26320.353,E2 -26320.353} C_VEL
LIN {X 0,Y 257.704,Z 339.368,A -85,B 0,C 180,E1 -26320.91,E2 -26320.91} C_VEL
LIN {X 0,Y 260.712,Z 344.148,A -85,B 0,C 180,E1 -26322.027,E2 -26322.027} C_VEL
LIN {X 0,Y 262.285,Z 346.432,A -85,B 0,C 180,E1 -26322.58,E2 -26322.58} C_VEL
LIN {X 0,Y 266.365,Z 352.946,A -85,B 0,C 180,E1 -26323.979,E2 -26323.979} C_VEL
LIN {X 0,Y 270.036,Z 359.051,A -85,B 0,C 180,E1 -26325.175,E2 -26325.175} C_VEL
LIN {X 0,Y 275.352,Z 368.222,A -85,B 0,C 180,E1 -26326.815,E2 -26326.815} C_VEL
LIN {X 0,Y 282.05,Z 381.023,A -85,B 0,C 180,E1 -26328.765,E2 -26328.765} C_VEL
LIN {X 0,Y 288.014,Z 394.014,A -85,B 0,C 180,E1 -26330.427,E2 -26330.427} C_VEL
LIN {X 0,Y 291.358,Z 402.348,A -85,B 0,C 180,E1 -26331.345,E2 -26331.345} C_VEL
LIN {X 0,Y 294.023,Z 424.167,A -85,B 0,C 180,E1 -26332.544,E2 -26332.544} C_VEL
LIN {X 0,Y 294.111,Z 428.68,A -85,B 0,C 180,E1 -26332.706,E2 -26332.706} C_VEL
LIN {X 0,Y 291.14,Z 480.992,A -85,B 0,C 180,E1 -26333.936,E2 -26333.936} C_VEL
LIN {X 0,Y 289.474,Z 495.378,A -85,B 0,C 180,E1 -26334.503,E2 -26334.503} C_VEL
LIN {X 0,Y 286.864,Z 509.768,A -85,B 0,C 180,E1 -26335.308,E2 -26335.308} C_VEL
LIN {X 0,Y 283.795,Z 522.57,A -85,B 0,C 180,E1 -26336.271,E2 -26336.271} C_VEL
LIN {X 0,Y 280.355,Z 535.018,A -85,B 0,C 180,E1 -26337.514,E2 -26337.514} C_VEL
LIN {X 0,Y 276.187,Z 547.583,A -85,B 0,C 180,E1 -26339.103,E2 -26339.103} C_VEL
LIN {X 0,Y 272.056,Z 559.011,A -85,B 0,C 180,E1 -26340.972,E2 -26340.972} C_VEL
LIN {X 0,Y 268.301,Z 568.166,A -85,B 0,C 180,E1 -26342.82,E2 -26342.82} C_VEL
LIN {X 0,Y 264.424,Z 576.699,A -85,B 0,C 180,E1 -26344.928,E2 -26344.928} C_VEL
LIN {X 0,Y 260.572,Z 584.905,A -85,B 0,C 180,E1 -26347.481,E2 -26347.481} C_VEL
LIN {X 0,Y 257.366,Z 591.556,A -85,B 0,C 180,E1 -26350.115,E2 -26350.115} C_VEL
LIN {X 0,Y 254.501,Z 597.515,A -85,B 0,C 180,E1 -26353.207,E2 -26353.207} C_VEL
LIN {X 0,Y 252.378,Z 601.834,A -85,B 0,C 180,E1 -26356.26,E2 -26356.26} C_VEL
LIN {X 0,Y 251.206,Z 604.371,A -85,B 0,C 180,E1 -26358.749,E2 -26358.749} C_VEL
LIN {X 0,Y 250.351,Z 606.389,A -85,B 0,C 180,E1 -26361.962,E2 -26361.962} C_VEL
LIN {X 0,Y 250.32,Z 607.112,A -85,B 0,C 180,E1 -26365.189,E2 -26365.189} C_VEL
LIN {X 0,Y 250.878,Z 606.755,A -85,B 0,C 180,E1 -26368.204,E2 -26368.204} C_VEL
LIN {X 0,Y 250.679,Z 611.538,A -85,B 0,C 180,E1 -26370.804,E2 -26370.804} C_VEL
LIN {X 0,Y 250.425,Z 614.9,A -85,B 0,C 180,E1 -26373.211,E2 -26373.211} C_VEL
LIN {X 0,Y 250.451,Z 618.128,A -85,B 0,C 180,E1 -26376.427,E2 -26376.427} C_VEL
LIN {X 0,Y 251.072,Z 620.008,A -85,B 0,C 180,E1 -26379.64,E2 -26379.64} C_VEL
LIN {X 0,Y 252.628,Z 620.611,A -85,B 0,C 180,E1 -26382.819,E2 -26382.819} C_VEL
LIN {X 0,Y 255.308,Z 619.848,A -85,B 0,C 180,E1 -26386.212,E2 -26386.212} C_VEL
LIN {X 0,Y 258.277,Z 618.022,A -85,B 0,C 180,E1 -26388.996,E2 -26388.996} C_VEL
LIN {X 0,Y 262.432,Z 614.804,A -85,B 0,C 180,E1 -26391.946,E2 -26391.946} C_VEL
LIN {X 0,Y 267.507,Z 610.21,A -85,B 0,C 180,E1 -26394.772,E2 -26394.772} C_VEL
LIN {X 0,Y 271.569,Z 605.799,A -85,B 0,C 180,E1 -26396.835,E2 -26396.835} C_VEL
LIN {X 0,Y 277.869,Z 598.533,A -85,B 0,C 180,E1 -26399.446,E2 -26399.446} C_VEL
LIN {X 0,Y 284.083,Z 590.647,A -85,B 0,C 180,E1 -26401.601,E2 -26401.601} C_VEL
LIN {X 0,Y 290.683,Z 581.121,A -85,B 0,C 180,E1 -26403.66,E2 -26403.66} C_VEL
LIN {X 0,Y 296.831,Z 571.307,A -85,B 0,C 180,E1 -26405.323,E2 -26405.323} C_VEL
LIN {X 0,Y 303.326,Z 559.633,A -85,B 0,C 180,E1 -26406.902,E2 -26406.902} C_VEL
LIN {X 0,Y 309.042,Z 547.949,A -85,B 0,C 180,E1 -26408.146,E2 -26408.146} C_VEL
LIN {X 0,Y 314.44,Z 535.361,A -85,B 0,C 180,E1 -26409.207,E2 -26409.207} C_VEL
LIN {X 0,Y 319.436,Z 521.496,A -85,B 0,C 180,E1 -26410.103,E2 -26410.103} C_VEL
LIN {X 0,Y 324.086,Z 505.58,A -85,B 0,C 180,E1 -26410.873,E2 -26410.873} C_VEL
LIN {X 0,Y 327.393,Z 490.124,A -85,B 0,C 180,E1 -26411.458,E2 -26411.458} C_VEL
LIN {X 0,Y 337.313,Z 434.57,A -85,B 0,C 180,E1 -26413.312,E2 -26413.312} C_VEL
LIN {X 0,Y 335.606,Z 430.721,A -85,B 0,C 180,E1 -26415.207,E2 -26415.207} C_VEL
LIN {X 0,Y 334.296,Z 428.338,A -85,B 0,C 180,E1 -26417.077,E2 -26417.077} C_VEL
LIN {X 0,Y 333.48,Z 426.604,A -85,B 0,C 180,E1 -26419.129,E2 -26419.129} C_VEL
LIN {X 0,Y 333.106,Z 426.448,A -85,B 0,C 180,E1 -26421.083,E2 -26421.083} C_VEL
LIN {X 0,Y 333.297,Z 427.752,A -85,B 0,C 180,E1 -26423.354,E2 -26423.354} C_VEL
LIN {X 0,Y 334.23,Z 430.585,A -85,B 0,C 180,E1 -26425.727,E2 -26425.727} C_VEL
LIN {X 0,Y 335.353,Z 434.274,A -85,B 0,C 180,E1 -26427.549,E2 -26427.549} C_VEL
LIN {X 0,Y 336.583,Z 438.514,A -85,B 0,C 180,E1 -26429.089,E2 -26429.089} C_VEL
LIN {X 0,Y 326.436,Z 494.4,A -85,B 0,C 180,E1 -26430.957,E2 -26430.957} C_VEL
LIN {X 0,Y 322.924,Z 508.387,A -85,B 0,C 180,E1 -26431.586,E2 -26431.586} C_VEL
LIN {X 0,Y 318.852,Z 521.347,A -85,B 0,C 180,E1 -26432.35,E2 -26432.35} C_VEL
LIN {X 0,Y 313.536,Z 535.621,A -85,B 0,C 180,E1 -26433.461,E2 -26433.461} C_VEL
LIN {X 0,Y 307.746,Z 548.484,A -85,B 0,C 180,E1 -26434.738,E2 -26434.738} C_VEL
LIN {X 0,Y 302.171,Z 559.259,A -85,B 0,C 180,E1 -26436.068,E2 -26436.068} C_VEL
LIN {X 0,Y 294.928,Z 571.516,A -85,B 0,C 180,E1 -26437.998,E2 -26437.998} C_VEL
LIN {X 0,Y 288.918,Z 580.436,A -85,B 0,C 180,E1 -26439.789,E2 -26439.789} C_VEL
LIN {X 0,Y 282.558,Z 588.905,A -85,B 0,C 180,E1 -26441.949,E2 -26441.949} C_VEL
LIN {X 0,Y 276.482,Z 596.058,A -85,B 0,C 180,E1 -26444.311,E2 -26444.311} C_VEL
LIN {X 0,Y 271.385,Z 601.353,A -85,B 0,C 180,E1 -26446.568,E2 -26446.568} C_VEL
LIN {X 0,Y 265.845,Z 606.247,A -85,B 0,C 180,E1 -26449.372,E2 -26449.372} C_VEL
LIN {X 0,Y 261.167,Z 609.655,A -85,B 0,C 180,E1 -26452.293,E2 -26452.293} C_VEL
LIN {X 0,Y 257.369,Z 611.685,A -85,B 0,C 180,E1 -26455.317,E2 -26455.317} C_VEL
LIN {X 0,Y 254.404,Z 612.405,A -85,B 0,C 180,E1 -26458.422,E2 -26458.422} C_VEL
LIN {X 0,Y 252.282,Z 611.788,A -85,B 0,C 180,E1 -26461.688,E2 -26461.688} C_VEL
LIN {X 0,Y 250.935,Z 609.929,A -85,B 0,C 180,E1 -26464.804,E2 -26464.804} C_VEL
LIN {X 0,Y 250.154,Z 606.66,A -85,B 0,C 180,E1 -26468.048,E2 -26468.048} C_VEL
LIN {X 0,Y 250.034,Z 603.219,A -85,B 0,C 180,E1 -26470.492,E2 -26470.492} C_VEL
LIN {X 0,Y 250.031,Z 598.84,A -85,B 0,C 180,E1 -26472.951,E2 -26472.951} C_VEL
LIN {X 0,Y 250.32,Z 592.377,A -85,B 0,C 180,E1 -26475.832,E2 -26475.832} C_VEL
LIN {X 0,Y 250.71,Z 584.401,A -85,B 0,C 180,E1 -26478.657,E2 -26478.657} C_VEL
LIN {X 0,Y 251.262,Z 575.409,A -85,B 0,C 180,E1 -26481.248,E2 -26481.248} C_VEL
LIN {X 0,Y 252,Z 564.533,A -85,B 0,C 180,E1 -26483.813,E2 -26483.813} C_VEL
LIN {X 0,Y 252.979,Z 552.758,A -85,B 0,C 180,E1 -26486.075,E2 -26486.075} C_VEL
LIN {X 0,Y 254.041,Z 540.062,A -85,B 0,C 180,E1 -26488.072,E2 -26488.072} C_VEL
LIN {X 0,Y 255.032,Z 527.972,A -85,B 0,C 180,E1 -26489.628,E2 -26489.628} C_VEL
LIN {X 0,Y 256.105,Z 513.908,A -85,B 0,C 180,E1 -26491.08,E2 -26491.08} C_VEL
LIN {X 0,Y 257.182,Z 498.628,A -85,B 0,C 180,E1 -26492.287,E2 -26492.287} C_VEL
LIN {X 0,Y 258.113,Z 483.244,A -85,B 0,C 180,E1 -26493.16,E2 -26493.16} C_VEL
LIN {X 0,Y 262.019,Z 389.036,A -85,B 0,C 180,E1 -26497.154,E2 -26497.154} C_VEL
LIN {X 0,Y 259.356,Z 361.624,A -85,B 0,C 180,E1 -26498.44,E2 -26498.44} C_VEL
LIN {X 0,Y 258.512,Z 351.064,A -85,B 0,C 180,E1 -26498.936,E2 -26498.936} C_VEL
LIN {X 0,Y 257.546,Z 346.977,A -85,B 0,C 180,E1 -26499.185,E2 -26499.185} C_VEL
LIN {X 0,Y 253.85,Z 328.525,A -85,B 0,C 180,E1 -26503.479,E2 -26503.479} C_VEL
LIN {X 0,Y 253.204,Z 325.499,A -85,B 0,C 180,E1 -26504.208,E2 -26504.208} C_VEL
LIN {X 0,Y 253.176,Z 325.506,A -85,B 0,C 180,E1 -26508.391,E2 -26508.391} C_VEL
LIN {X 0,Y 253.137,Z 325.511,A -85,B 0,C 180,E1 -26512.497,E2 -26512.497} C_VEL
LIN {X 0,Y 253.218,Z 325.482,A -85,B 0,C 180,E1 -26516.407,E2 -26516.407} C_VEL
LIN {X 0,Y 253.144,Z 325.507,A -85,B 0,C 180,E1 -26520.125,E2 -26520.125} C_VEL
LIN {X 0,Y 253.204,Z 325.499,A -85,B 0,C 180,E1 -26523.726,E2 -26523.726} C_VEL
LIN {X 0,Y 253.283,Z 325.493,A -85,B 0,C 180,E1 -26528.075,E2 -26528.075} C_VEL
LIN {X 0,Y 253.303,Z 325.524,A -85,B 0,C 180,E1 -26528.596,E2 -26528.596} C_VEL
LIN {X 0,Y 254.259,Z 328.263,A -85,B 0,C 180,E1 -26528.802,E2 -26528.802} C_VEL
LIN {X 0,Y 261.682,Z 342.841,A -85,B 0,C 180,E1 -26530.135,E2 -26530.135} C_VEL
LIN {X 0,Y 269.869,Z 361.502,A -85,B 0,C 180,E1 -26531.578,E2 -26531.578} C_VEL
LIN {X 0,Y 271.252,Z 365.565,A -85,B 0,C 180,E1 -26531.838,E2 -26531.838} C_VEL
LIN {X 0,Y 268.092,Z 453.599,A -85,B 0,C 180,E1 -26534.123,E2 -26534.123} C_VEL
LIN {X 0,Y 267.151,Z 467.283,A -85,B 0,C 180,E1 -26534.748,E2 -26534.748} C_VEL
LIN {X 0,Y 266.04,Z 480.157,A -85,B 0,C 180,E1 -26535.609,E2 -26535.609} C_VEL
LIN {X 0,Y 264.506,Z 493.402,A -85,B 0,C 180,E1 -26536.794,E2 -26536.794} C_VEL
LIN {X 0,Y 262.751,Z 504.796,A -85,B 0,C 180,E1 -26538.073,E2 -26538.073} C_VEL
LIN {X 0,Y 260.633,Z 516.7,A -85,B 0,C 180,E1 -26539.74,E2 -26539.74} C_VEL
LIN {X 0,Y 258.617,Z 528.483,A -85,B 0,C 180,E1 -26541.822,E2 -26541.822} C_VEL
LIN {X 0,Y 256.508,Z 539.048,A -85,B 0,C 180,E1 -26544.119,E2 -26544.119} C_VEL
LIN {X 0,Y 254.788,Z 547.765,A -85,B 0,C 180,E1 -26546.45,E2 -26546.45} C_VEL
LIN {X 0,Y 253.235,Z 555.04,A -85,B 0,C 180,E1 -26548.807,E2 -26548.807} C_VEL
LIN {X 0,Y 252.262,Z 562.05,A -85,B 0,C 180,E1 -26551.627,E2 -26551.627} C_VEL
LIN {X 0,Y 251.505,Z 566.789,A -85,B 0,C 180,E1 -26553.989,E2 -26553.989} C_VEL
LIN {X 0,Y 250.695,Z 571.817,A -85,B 0,C 180,E1 -26557.219,E2 -26557.219} C_VEL
LIN {X 0,Y 250.468,Z 574.598,A -85,B 0,C 180,E1 -26559.655,E2 -26559.655} C_VEL
LIN {X 0,Y 250.485,Z 577.058,A -85,B 0,C 180,E1 -26562.923,E2 -26562.923} C_VEL
LIN {X 0,Y 250.925,Z 578.162,A -85,B 0,C 180,E1 -26566.205,E2 -26566.205} C_VEL
LIN {X 0,Y 251.946,Z 577.907,A -85,B 0,C 180,E1 -26569.484,E2 -26569.484} C_VEL
LIN {X 0,Y 253.459,Z 576.283,A -85,B 0,C 180,E1 -26572.757,E2 -26572.757} C_VEL
LIN {X 0,Y 255.71,Z 573.23,A -85,B 0,C 180,E1 -26575.989,E2 -26575.989} C_VEL
LIN {X 0,Y 257.785,Z 569.899,A -85,B 0,C 180,E1 -26578.387,E2 -26578.387} C_VEL
LIN {X 0,Y 260.238,Z 565.663,A -85,B 0,C 180,E1 -26580.752,E2 -26580.752} C_VEL
LIN {X 0,Y 263.629,Z 559.399,A -85,B 0,C 180,E1 -26583.452,E2 -26583.452} C_VEL
LIN {X 0,Y 267.382,Z 551.764,A -85,B 0,C 180,E1 -26586.018,E2 -26586.018} C_VEL
LIN {X 0,Y 271.227,Z 543.207,A -85,B 0,C 180,E1 -26588.296,E2 -26588.296} C_VEL
LIN {X 0,Y 275.006,Z 533.999,A -85,B 0,C 180,E1 -26590.267,E2 -26590.267} C_VEL
LIN {X 0,Y 278.951,Z 522.914,A -85,B 0,C 180,E1 -26592.192,E2 -26592.192} C_VEL
LIN {X 0,Y 282.824,Z 510.47,A -85,B 0,C 180,E1 -26593.898,E2 -26593.898} C_VEL
LIN {X 0,Y 286.013,Z 497.984,A -85,B 0,C 180,E1 -26595.246,E2 -26595.246} C_VEL
LIN {X 0,Y 288.608,Z 485.105,A -85,B 0,C 180,E1 -26596.342,E2 -26596.342} C_VEL
LIN {X 0,Y 290.85,Z 470.942,A -85,B 0,C 180,E1 -26597.231,E2 -26597.231} C_VEL
LIN {X 0,Y 292.296,Z 457.482,A -85,B 0,C 180,E1 -26597.829,E2 -26597.829} C_VEL
LIN {X 0,Y 293.508,Z 436.582,A -85,B 0,C 180,E1 -26598.392,E2 -26598.392} C_VEL
LIN {X 0,Y 295.886,Z 392.437,A -85,B 0,C 180,E1 -26599.408,E2 -26599.408} C_VEL
LIN {X 0,Y 289.558,Z 379.342,A -85,B 0,C 180,E1 -26601.028,E2 -26601.028} C_VEL
LIN {X 0,Y 282.293,Z 367.019,A -85,B 0,C 180,E1 -26602.942,E2 -26602.942} C_VEL
LIN {X 0,Y 274.653,Z 355.28,A -85,B 0,C 180,E1 -26605.101,E2 -26605.101} C_VEL
LIN {X 0,Y 269.957,Z 348.507,A -85,B 0,C 180,E1 -26606.525,E2 -26606.525} C_VEL
LIN {X 0,Y 266.43,Z 343.772,A -85,B 0,C 180,E1 -26607.643,E2 -26607.643} C_VEL
LIN {X 0,Y 263.626,Z 339.996,A -85,B 0,C 180,E1 -26608.575,E2 -26608.575} C_VEL
LIN {X 0,Y 261.118,Z 336.479,A -85,B 0,C 180,E1 -26609.45,E2 -26609.45} C_VEL
LIN {X 0,Y 258.053,Z 332.952,A -85,B 0,C 180,E1 -26610.531,E2 -26610.531} C_VEL
LIN {X 0,Y 256.993,Z 330.945,A -85,B 0,C 180,E1 -26610.956,E2 -26610.956} C_VEL
LIN {X 0,Y 254.6,Z 328.957,A -85,B 0,C 180,E1 -26611.819,E2 -26611.819} C_VEL
LIN {X 0,Y 253.414,Z 326.551,A -85,B 0,C 180,E1 -26612.333,E2 -26612.333} C_VEL
LIN {X 0,Y 253.222,Z 325.487,A -85,B 0,C 180,E1 -26612.512,E2 -26612.512} C_VEL
LIN {X 0,Y 253.211,Z 325.486,A -85,B 0,C 180,E1 -26617.215,E2 -26617.215} C_VEL
LIN {X 0,Y 253.314,Z 325.472,A -85,B 0,C 180,E1 -26620.621,E2 -26620.621} C_VEL
LIN {X 0,Y 253.402,Z 325.458,A -85,B 0,C 180,E1 -26625.595,E2 -26625.595} C_VEL
LIN {X 0,Y 253.49,Z 325.446,A -85,B 0,C 180,E1 -26630.457,E2 -26630.457} C_VEL
LIN {X 0,Y 253.71,Z 325.441,A -85,B 0,C 180,E1 -26633.66,E2 -26633.66} C_VEL
LIN {X 0,Y 253.797,Z 325.424,A -85,B 0,C 180,E1 -26638.419,E2 -26638.419} C_VEL
LIN {X 0,Y 253.918,Z 325.406,A -85,B 0,C 180,E1 -26640,E2 -26640} C_VEL
LIN {X 0,Y 253.728,Z 325.438,A -85,B 0,C 180,E1 -26644.751,E2 -26644.751} C_VEL
LIN {X 0,Y 253.561,Z 325.434,A -85,B 0,C 180,E1 -26647.939,E2 -26647.939} C_VEL
LIN {X 0,Y 253.415,Z 325.45,A -85,B 0,C 180,E1 -26652.775,E2 -26652.775} C_VEL
LIN {X 0,Y 253.31,Z 325.475,A -85,B 0,C 180,E1 -26656.052,E2 -26656.052} C_VEL
LIN {X 0,Y 253.305,Z 325.488,A -85,B 0,C 180,E1 -26659.933,E2 -26659.933} C_VEL
LIN {X 0,Y 253.211,Z 325.502,A -85,B 0,C 180,E1 -26664.515,E2 -26664.515} C_VEL
LIN {X 0,Y 253.193,Z 325.499,A -85,B 0,C 180,E1 -26668.054,E2 -26668.054} C_VEL
LIN {X 0,Y 253.167,Z 325.495,A -85,B 0,C 180,E1 -26671.006,E2 -26671.006} C_VEL
LIN {X 0,Y 252.945,Z 325.92,A -85,B 0,C 180,E1 -26671.889,E2 -26671.889} C_VEL
LIN {X 0,Y 252.104,Z 327.721,A -85,B 0,C 180,E1 -26673.159,E2 -26673.159} C_VEL
LIN {X 0,Y 249.799,Z 333.984,A -85,B 0,C 180,E1 -26675.991,E2 -26675.991} C_VEL
LIN {X 0,Y 249.612,Z 336.465,A -85,B 0,C 180,E1 -26677.244,E2 -26677.244} C_VEL
LIN {X 0,Y 249.773,Z 337.188,A -85,B 0,C 180,E1 -26677.671,E2 -26677.671} C_VEL
LIN {X 0,Y 250.265,Z 338.651,A -85,B 0,C 180,E1 -26678.458,E2 -26678.458} C_VEL
LIN {X 0,Y 253.454,Z 343.615,A -85,B 0,C 180,E1 -26679.776,E2 -26679.776} C_VEL
LIN {X 0,Y 255.04,Z 345.85,A -85,B 0,C 180,E1 -26680.391,E2 -26680.391} C_VEL
LIN {X 0,Y 259.204,Z 352.275,A -85,B 0,C 180,E1 -26681.956,E2 -26681.956} C_VEL
LIN {X 0,Y 263.152,Z 358.641,A -85,B 0,C 180,E1 -26683.357,E2 -26683.357} C_VEL
LIN {X 0,Y 268.697,Z 368.036,A -85,B 0,C 180,E1 -26685.205,E2 -26685.205} C_VEL
LIN {X 0,Y 275.835,Z 381.367,A -85,B 0,C 180,E1 -26687.427,E2 -26687.427} C_VEL
LIN {X 0,Y 282.34,Z 395.252,A -85,B 0,C 180,E1 -26689.337,E2 -26689.337} C_VEL
LIN {X 0,Y 286.391,Z 405.219,A -85,B 0,C 180,E1 -26690.498,E2 -26690.498} C_VEL
LIN {X 0,Y 288.894,Z 426.621,A -85,B 0,C 180,E1 -26691.703,E2 -26691.703} C_VEL
LIN {X 0,Y 285.926,Z 479.282,A -85,B 0,C 180,E1 -26692.96,E2 -26692.96} C_VEL
LIN {X 0,Y 284.217,Z 494.08,A -85,B 0,C 180,E1 -26693.525,E2 -26693.525} C_VEL
LIN {X 0,Y 281.864,Z 507.55,A -85,B 0,C 180,E1 -26694.274,E2 -26694.274} C_VEL
LIN {X 0,Y 278.929,Z 519.867,A -85,B 0,C 180,E1 -26695.164,E2 -26695.164} C_VEL
LIN {X 0,Y 275.265,Z 532.764,A -85,B 0,C 180,E1 -26696.401,E2 -26696.401} C_VEL
LIN {X 0,Y 270.97,Z 545.649,A -85,B 0,C 180,E1 -26698.005,E2 -26698.005} C_VEL
LIN {X 0,Y 267.063,Z 556.196,A -85,B 0,C 180,E1 -26699.681,E2 -26699.681} C_VEL
LIN {X 0,Y 262.811,Z 566.45,A -85,B 0,C 180,E1 -26701.704,E2 -26701.704} C_VEL
LIN {X 0,Y 258.631,Z 575.402,A -85,B 0,C 180,E1 -26703.895,E2 -26703.895} C_VEL
LIN {X 0,Y 254.543,Z 583.792,A -85,B 0,C 180,E1 -26706.488,E2 -26706.488} C_VEL
LIN {X 0,Y 251.512,Z 589.671,A -85,B 0,C 180,E1 -26708.779,E2 -26708.779} C_VEL
LIN {X 0,Y 248.363,Z 596.01,A -85,B 0,C 180,E1 -26711.932,E2 -26711.932} C_VEL
LIN {X 0,Y 245.911,Z 600.761,A -85,B 0,C 180,E1 -26715.151,E2 -26715.151} C_VEL
LIN {X 0,Y 244.228,Z 604.058,A -85,B 0,C 180,E1 -26718.423,E2 -26718.423} C_VEL
LIN {X 0,Y 243.317,Z 606.015,A -85,B 0,C 180,E1 -26721.729,E2 -26721.729} C_VEL
LIN {X 0,Y 243.224,Z 606.682,A -85,B 0,C 180,E1 -26725.048,E2 -26725.048} C_VEL
LIN {X 0,Y 243.849,Z 606.031,A -85,B 0,C 180,E1 -26728.461,E2 -26728.461} C_VEL
LIN {X 0,Y 243.694,Z 610.372,A -85,B 0,C 180,E1 -26730.827,E2 -26730.827} C_VEL
LIN {X 0,Y 243.396,Z 613.951,A -85,B 0,C 180,E1 -26733.304,E2 -26733.304} C_VEL
LIN {X 0,Y 243.424,Z 617.417,A -85,B 0,C 180,E1 -26736.613,E2 -26736.613} C_VEL
LIN {X 0,Y 244.068,Z 619.529,A -85,B 0,C 180,E1 -26739.919,E2 -26739.919} C_VEL
LIN {X 0,Y 245.714,Z 620.386,A -85,B 0,C 180,E1 -26743.186,E2 -26743.186} C_VEL
LIN {X 0,Y 248.243,Z 619.986,A -85,B 0,C 180,E1 -26746.393,E2 -26746.393} C_VEL
LIN {X 0,Y 251.574,Z 618.341,A -85,B 0,C 180,E1 -26749.522,E2 -26749.522} C_VEL
LIN {X 0,Y 255.885,Z 615.421,A -85,B 0,C 180,E1 -26752.538,E2 -26752.538} C_VEL
LIN {X 0,Y 261.155,Z 611.14,A -85,B 0,C 180,E1 -26755.416,E2 -26755.416} C_VEL
LIN {X 0,Y 265.36,Z 607.07,A -85,B 0,C 180,E1 -26757.515,E2 -26757.515} C_VEL
LIN {X 0,Y 271.848,Z 600.193,A -85,B 0,C 180,E1 -26760.165,E2 -26760.165} C_VEL
LIN {X 0,Y 279.193,Z 591.528,A -85,B 0,C 180,E1 -26762.646,E2 -26762.646} C_VEL
LIN {X 0,Y 285.018,Z 583.71,A -85,B 0,C 180,E1 -26764.422,E2 -26764.422} C_VEL
LIN {X 0,Y 291.344,Z 574.481,A -85,B 0,C 180,E1 -26766.091,E2 -26766.091} C_VEL
LIN {X 0,Y 298.008,Z 563.52,A -85,B 0,C 180,E1 -26767.673,E2 -26767.673} C_VEL
LIN {X 0,Y 303.793,Z 552.719,A -85,B 0,C 180,E1 -26768.928,E2 -26768.928} C_VEL
LIN {X 0,Y 309.93,Z 539.717,A -85,B 0,C 180,E1 -26770.102,E2 -26770.102} C_VEL
LIN {X 0,Y 315.26,Z 526.316,A -85,B 0,C 180,E1 -26771.04,E2 -26771.04} C_VEL
LIN {X 0,Y 320.615,Z 509.937,A -85,B 0,C 180,E1 -26771.893,E2 -26771.893} C_VEL
